# B&R Automation Studio project 8238 (part 7)

#### zz_KanlinkConfig.ab - Implementation code
```automation-basic
(********************************************************************
 * COPYRIGHT -- HP
 ********************************************************************
 * Program: zz_KanlinkConfig
 * File: zz_KanlinkConfig.ab
 * Author: treamsbottom
 * Created: September 07, 2012
 ********************************************************************
 * Implementation of program zz_KanlinkConfig
 ********************************************************************)
;Requirements
;From KGFramework
;	Libaries:
;		KgStdLib
;		KanLinkLib
;		mnParamLib
;	10ms Tasks:
;		hlKanLink
;	100ms Tasks:
;		svCPCache
;		mnEth
; When setting max connections for anything greater than 10
;the array decs will need changing. these are set by the constants HLKANLINK_MAX_CLIENTCONNS and HLKANLINK_MAX_SERVERCONNS in the frameworkshare
;Pkg_hlKanLink, KL_UserLib.Var
;----------------------------------------------------------------------------------------------------------------;
;-----21-1-2013..TR..Version A6 - First TestedVersion - Note Specials to run with Shuttle
;-----28-1-2013..TR..Version A7 - Remove Specials..Add option to send program and category number & Batch number.#
;-----03-03-2017..TR.Version A18 - Add "Advanced Connection Mode"
;-----07-06-2017 ..TR..Version A19 - Fix issues with sending empty bag date-- Remove reference to CAN[].Category -- Read all information from bag for consistency.
;-----------------------------------------------------------------------------------------------------------------
PROGRAM _INIT
	init := 0;
END_PROGRAM
PROGRAM _CYCLIC
;HLKANLINK_MAX_SERVERCONNS	;Declaration of max Server conns for KG Framework
;HLKANLINK_MAX_CLIENTCONNS	;Declaration of max Client conns for KG Framework
IF NOT init THEN
;Parameter Setup
;Global setting - Apply to all Kanlink Comms(Server,Client,OverView)
	Kanlink.GlobalSettings.TransferProgramCode 	= FALSE ; This transfers/Read the cat code to/from the bCustom area. Prg to/from sCategory
	Kanlink.GlobalSettings.TransferProgin_bCustom = FALSE ;This transfers/Read the Program code to/from the bCustom area. Category to/from sCategory
	Kanlink.GlobalSettings.UseBatchCode 		= TRUE	; Pass batch/SQL id
	Kanlink.GlobalSettings.BatchCodeTyp			= BatchTyp_UDINT  ;0 = UDINT, 1 = 16 byte unique (UDINT By default, extra code required for 16 byte )

;---------------------------------------------------------Batch Transfer Server---------------------------------------------------------------
;Server (Used to send data)		--------------------------- Variable = PT100
	Kanlink.Server.Enable = TRUE ; used to enable Server Comms
	Kanlink.Server.MaxConns	= 1 ; Number of Server connections
	 ; Start address of CAN variable
	;Address
	Kanlink.Server.IP[1].CommID = 1; //SDC1 R43
	Kanlink.Server.IP[1].Area 	= 3
	Kanlink.Server.IP[1].Adr 	= 11
;	Kanlink.Server.IP[1].AdvMode = FALSE // Use Advance mode- Pass in whole IP address as a string.
;	strcpy(ADR(Kanlink.Server.IP[1].AdrAdvMode),ADR("10.8.3.13"));
	Kanlink.Server.IP[1].CmdOpt = 0;

;	Kanlink.Server.IP[2].CommID = 2; //SDC2 R45
;	Kanlink.Server.IP[2].Area 	= 3
;	Kanlink.Server.IP[2].Adr 	= 12
;	Kanlink.Server.IP[2].CmdOpt = 0;
;
;	Kanlink.Server.IP[3].CommID = 3; //SDC3 R47
;	Kanlink.Server.IP[3].Area 	= 3
;	Kanlink.Server.IP[3].Adr 	= 13
;	Kanlink.Server.IP[3].CmdOpt = 0;
;
;	Kanlink.Server.IP[4].CommID = 4; //CDC8 R110
;	Kanlink.Server.IP[4].Area 	= 1
;	Kanlink.Server.IP[4].Adr 	= 12
;	Kanlink.Server.IP[4].CmdOpt = 0;
;
;	Kanlink.Server.IP[5].CommID = 5; //CDC9 R113
;	Kanlink.Server.IP[5].Area 	= 1
;	Kanlink.Server.IP[5].Adr 	= 2
;	Kanlink.Server.IP[5].CmdOpt = 0;
;
;	Kanlink.Server.IP[6].CommID = 6; //CDC6 R68
;	Kanlink.Server.IP[6].Area 	= 5
;	Kanlink.Server.IP[6].Adr 	= 15
;	Kanlink.Server.IP[6].CmdOpt = 0;
;
;	Kanlink.Server.IP[7].CommID = 7; //CDC7 R70
;	Kanlink.Server.IP[7].Area 	= 5
;	Kanlink.Server.IP[7].Adr 	= 16
;	Kanlink.Server.IP[7].CmdOpt = 0;
	;---------------------------------------------------------Batch transfer Client---------------------------------------------------------------
	;Client used to recieve data --------------------------- Variable = PTResp
	Kanlink.Client.Enable = TRUE ; used to enable Client Comms
	Kanlink.Client.MaxConns	= 2 ; Number of Client connections
	;Address

	//CSL1 r41
	Kanlink.Client.IP[1].CommID = 14	;//CSL1
	Kanlink.Client.IP[1].Area 	= 3
	Kanlink.Client.IP[1].Adr 	= 64
;	Kanlink.Client.IP[1].AdvMode = FALSE // Use Advance mode- Pass in whole IP address as a string.
;	strcpy(ADR(Kanlink.Client.IP[1].AdrAdvMode),ADR("10.8.4.20"));
	Kanlink.Client.IP[1].CmdOpt = 0

	//CSL2 r43
	Kanlink.Client.IP[2].CommID = 15	;//CSL2
	Kanlink.Client.IP[2].Area 	= 3
	Kanlink.Client.IP[2].Adr 	= 64
	Kanlink.Client.IP[2].CmdOpt = 1
;
;	//CSL1 r49
;	Kanlink.Client.IP[3].CommID = 11	;//CSL3
;	Kanlink.Client.IP[3].Area 	= 3
;	Kanlink.Client.IP[3].Adr 	= 62
;	Kanlink.Client.IP[3].CmdOpt = 0

;	//Sorting Rail
;	Kanlink.Client.IP[2].CommID = 4
;	Kanlink.Client.IP[2].Area 	= 3 ;Aero at sorting
;	Kanlink.Client.IP[2].Adr 	= 64
	;	Kanlink.Client.IP[1].AdvMode = FALSE // Use Advance mode- Pass in whole IP address as a string.
	;	strcpy(ADR(Kanlink.Client.IP[1].AdrAdvMode),ADR("10.8.4.20"));
;	Kanlink.Client.IP[2].CmdOpt = 1
;

;;---------------------------------------------------------Overview Server---------------------------------------------------------------
;	;------------------------------------------------Variable = STOverResp
;	;Use Overview Server.. SendData Data to Overview PLC - Only IP necessary - Client will request bag numbers.
	Kanlink.OverviewServer.Enable = FALSE
;	Kanlink.OverviewServer.MaxConns = 1
;
;	Kanlink.OverviewServer.IP[1].Area = 4
;	Kanlink.OverviewServer.IP[1].Adr = 21
;	Kanlink.OverviewServer.IP[1].AdvMode = FALSE
;	strcpy(ADR(Kanlink.OverviewServer.IP[1].AdrAdvMode),ADR("10.8.2.21"));
;
;	Kanlink.OverviewServer.IP[1].CmdOpt = 0
;;---------------------------------------------------------Overview Client---------------------------------------------------------------
;;------------------------------------------------Variable = STOverReq
;;Use Overview Client.. Recieve Data
	Kanlink.OverviewClient.Enable = FALSE
;	Kanlink.OverviewClient.MaxConns = 5
;	Kanlink.OverviewClient.CANOffset = 21
;;-----------PLC 1 - AERO SYSTEM
;	Kanlink.OverviewClient.StatusReg[1] = 951 ; D reg to map machine status for Tview.
;
;
;	Kanlink.OverviewClient.IP[1].Area = 3
;	Kanlink.OverviewClient.IP[1].Adr = 1	; To multiplex Edit KL_Overview
;	Kanlink.OverviewClient.IP[1].AdvMode = FALSE
;	strcpy(ADR(Kanlink.OverviewClient.IP[1].AdrAdvMode),ADR("10.8.3.1"));
;
;	Kanlink.OverviewClient.IP[1].CmdOpt = 0
;	//Batch data requested from Server
;	Kanlink.OverviewClient.InfoReq[1].wCntPositions = 6  ;Number of positions requested max 6 per request. If more than 6 set to 0 to multiplex...
;	Kanlink.OverviewClient.InfoReq[1].wNoOfPosition[0] = 1  ; Unqiue ID of data requested put all requests here if more than 6 the driver will multiplex the signals.
;	Kanlink.OverviewClient.InfoReq[1].wNoOfPosition[1] = 2	; There must be no gaps in the request numbers.	If not multiplexing, ensure index[6] = 0
;	Kanlink.OverviewClient.InfoReq[1].wNoOfPosition[2] = 3
;	Kanlink.OverviewClient.InfoReq[1].wNoOfPosition[3] = 4
;	Kanlink.OverviewClient.InfoReq[1].wNoOfPosition[4] = 5
;	Kanlink.OverviewClient.InfoReq[1].wNoOfPosition[5] = 6
;
;	//Bag number to map recieved data to.
;	Kanlink.OverviewClient.InfoResp[1].BagNum[0] = 501
;	Kanlink.OverviewClient.InfoResp[1].BagNum[1] = 502
;	Kanlink.OverviewClient.InfoResp[1].BagNum[2] = 503
;	Kanlink.OverviewClient.InfoResp[1].BagNum[3] = 504
;	Kanlink.OverviewClient.InfoResp[1].BagNum[4] = 505
;	Kanlink.OverviewClient.InfoResp[1].BagNum[5] = 506

;--------------------------------------------------------------END OF Configuration Code--------------------------------------------

;Check size of server and Client
	IF NOT Kanlink.Server.Enable THEN
		Kanlink.Server.MaxConns = 0
	ENDIF
	IF NOT Kanlink.Client.Enable THEN
		Kanlink.Client.MaxConns = 0
	ENDIF
	IF NOT Kanlink.OverviewServer.Enable THEN
		Kanlink.OverviewServer.MaxConns = 0
	ENDIF
	IF NOT Kanlink.OverviewClient.Enable THEN
		Kanlink.OverviewClient.MaxConns = 0
	ENDIF
	IF ((Kanlink.Server.MaxConns + Kanlink.OverviewServer.MaxConns) <= HLKANLINK_MAX_SERVERCONNS) THEN
		ServerDecOK = TRUE
	ELSE
		strcpy(ADR(Kanlink.ErrorString),"Declaration of HLKANLINK_MAX_SERVERCONNS not large enough")
		ServerDecOK = FALSE
	ENDIF
	IF ((Kanlink.Client.MaxConns + Kanlink.OverviewClient.MaxConns) <= HLKANLINK_MAX_CLIENTCONNS) THEN
		ClientDecOK = TRUE
	ELSE
		ClientDecOK = FALSE
		strcpy(ADR(Kanlink.ErrorString),"Declaration of HLKANLINK_MAX_CLIENTCONNS not large enough")
	ENDIF

	IF 	ServerDecOK AND ClientDecOK THEN

		;Server init
		IF Kanlink.Server.Enable THEN
			LOOP n = 1 TO Kanlink.Server.MaxConns DO
				;Build strings to pass to variable names, only required in a loop as index number changes.
				itoa(n,ADR(sn))	; put n into string
				strcpy(ADR(sReq),"PT100[");build string for variable name (request)
				strcat(ADR(sReq),ADR(sn))
				strcat(ADR(sReq),"].Req")
				strcpy(ADR(sResp),"PT100[");;build string for variable name (response)
				strcat(ADR(sResp),ADR(sn))
				strcat(ADR(sResp),"].Resp")
				IF Kanlink.Server.IP[n].AdvMode THEN
					IFhlKanLink.Parameter.Server[n].Adr = 0;
					IFhlKanLink.Parameter.Server[n].Area = 0
					IFhlKanLink.Parameter.Server[n].AdvMode := TRUE;
					strcpy(ADR(IFhlKanLink.Parameter.Server[n].AdrAdvMode),ADR(Kanlink.Server.IP[n].AdrAdvMode));
				ELSE
					IFhlKanLink.Parameter.Server[n].Adr = Kanlink.Server.IP[n].Adr ; Populate these arrays .
					IFhlKanLink.Parameter.Server[n].Area = Kanlink.Server.IP[n].Area
				ENDIF
				IFhlKanLink.Parameter.Server[n].Cmd = 1000 ; cmd from the server are always even
				IFhlKanLink.Parameter.Server[n].CmdOpt = Kanlink.Server.IP[n].CmdOpt
				IFhlKanLink.Parameter.Server[n].TimeOut = 1000 ;ms
				strcpy(ADR(IFhlKanLink.Parameter.Server[n].Name),"PT100") ; Diags Only
				strcpy(ADR(IFhlKanLink.Parameter.Server[n].sReq),ADR(sReq));"zzKanLink:PT100[0].Req")
				strcpy(ADR(IFhlKanLink.Parameter.Server[n].sResp),ADR(sResp));"zzKanLink:PT100[0].Resp")
			ENDLOOP
		ENDIF
		;Client Init
		IF Kanlink.Client.Enable THEN
			LOOP n = 1 TO Kanlink.Client.MaxConns DO
				itoa(n,ADR(sn))	; put n into string
				strcpy(ADR(sReq),"PTResp[");build string for variable name (request)
				strcat(ADR(sReq),ADR(sn))
				strcat(ADR(sReq),"].Req")
				strcpy(ADR(sResp),"PTResp[");;build string for variable name (response)
				strcat(ADR(sResp),ADR(sn))
				strcat(ADR(sResp),"].Resp")

				IF Kanlink.Client.IP[n].AdvMode THEN
					IFhlKanLink.Parameter.Client[n].Adr = 0;
					IFhlKanLink.Parameter.Client[n].Area = 0
					IFhlKanLink.Parameter.Client[n].AdvMode := TRUE;
					strcpy(ADR(IFhlKanLink.Parameter.Client[n].AdrAdvMode),ADR(Kanlink.Client.IP[n].AdrAdvMode));
				ELSE
					IFhlKanLink.Parameter.Client[n].Adr = Kanlink.Client.IP[n].Adr ; Populate these arrays .
					IFhlKanLink.Parameter.Client[n].Area = Kanlink.Client.IP[n].Area
				ENDIF
				IFhlKanLink.Parameter.Client[n].Cmd = 1000
				IFhlKanLink.Parameter.Client[n].CmdOpt = Kanlink.Client.IP[n].CmdOpt
				IFhlKanLink.Parameter.Client[n].CycleTime = 1000;ms
				strcpy(ADR(IFhlKanLink.Parameter.Client[n].Name),"PTResp")
				strcpy(ADR(IFhlKanLink.Parameter.Client[n].sReq),ADR(sReq))
				strcpy(ADR(IFhlKanLink.Parameter.Client[n].sResp),ADR(sResp))
			ENDLOOP
		ENDIF
		;Overview Server init
		;STOverResp[0] //Server sends batch data...
		IF Kanlink.OverviewServer.Enable THEN
			LOOP n = 1 TO Kanlink.OverviewServer.MaxConns DO
				;Build strings to pass to variable names, only required in a loop as index number changes.
				itoa(n,ADR(sn))	; put n into string
				strcpy(ADR(sReq),"STOverResp[");build string for variable name (request)
				strcat(ADR(sReq),ADR(sn))
				strcat(ADR(sReq),"].Req")
				strcpy(ADR(sResp),"STOverResp[");;build string for variable name (response)
				strcat(ADR(sResp),ADR(sn))
				strcat(ADR(sResp),"].Resp")

				Index = n + Kanlink.Server.MaxConns
				Kanlink.OverviewServer.IndexOffset = Kanlink.Server.MaxConns
				IF Kanlink.OverviewServer.IP[n].AdvMode THEN
					IFhlKanLink.Parameter.Server[Index].Adr = 0;
					IFhlKanLink.Parameter.Server[Index].Area = 0
					IFhlKanLink.Parameter.Server[Index].AdvMode := TRUE;
					strcpy(ADR(IFhlKanLink.Parameter.Server[Index].AdrAdvMode),ADR(Kanlink.OverviewServer.IP[n].AdrAdvMode));
				ELSE
					IFhlKanLink.Parameter.Server[Index].Adr = Kanlink.OverviewServer.IP[n].Adr ; Populate these arrays .
					IFhlKanLink.Parameter.Server[Index].Area = Kanlink.OverviewServer.IP[n].Area
				ENDIF

				IFhlKanLink.Parameter.Server[Index].Cmd = 1002 ;Batch Info Command
				IFhlKanLink.Parameter.Server[Index].CmdOpt = Kanlink.OverviewServer.IP[n].CmdOpt
				IFhlKanLink.Parameter.Server[Index].TimeOut = 1000 ;ms
				strcpy(ADR(IFhlKanLink.Parameter.Server[Index].Name),"STOverResp") ; Diags Only
				strcpy(ADR(IFhlKanLink.Parameter.Server[Index].sReq),ADR(sReq));"zzKanLink:STOverReq[0].Req")
				strcpy(ADR(IFhlKanLink.Parameter.Server[Index].sResp),ADR(sResp));"zzKanLink:STOverReq[0].Resp")

			ENDLOOP
		ENDIF

		;Kanlink OverView Client
		;STOverReq[0]// Client recieves batch data
		IF Kanlink.OverviewClient.Enable THEN
			LOOP n = 1 TO Kanlink.OverviewClient.MaxConns DO
				;Build strings to pass to variable names, only required in a loop as index number changes.
				itoa(n,ADR(sn))	; put n into string
				strcpy(ADR(sReq),"STOverReq[");build string for variable name (request)
				strcat(ADR(sReq),ADR(sn))
				strcat(ADR(sReq),"].Req")
				strcpy(ADR(sResp),"STOverReq[");;build string for variable name (response)
				strcat(ADR(sResp),ADR(sn))
				strcat(ADR(sResp),"].Resp")
				Index = n + Kanlink.Client.MaxConns
				Kanlink.OverviewClient.IndexOffset = Kanlink.Client.MaxConns

				IF Kanlink.OverviewClient.IP[n].AdvMode THEN
					IFhlKanLink.Parameter.Client[Index].Adr = 0;
					IFhlKanLink.Parameter.Client[Index].Area = 0
					IFhlKanLink.Parameter.Client[Index].AdvMode := TRUE;
					strcpy(ADR(IFhlKanLink.Parameter.Server[Index].AdrAdvMode),ADR(Kanlink.OverviewClient.IP[n].AdrAdvMode));
				ELSE
					IFhlKanLink.Parameter.Client[Index].Adr = Kanlink.OverviewClient.IP[n].Adr ; Populate these arrays .
					IFhlKanLink.Parameter.Client[Index].Area = Kanlink.OverviewClient.IP[n].Area
				ENDIF

				IFhlKanLink.Parameter.Client[Index].Cmd = 1002 ;Batch Info Command
				IFhlKanLink.Parameter.Client[Index].CmdOpt = Kanlink.OverviewClient.IP[n].CmdOpt
				IFhlKanLink.Parameter.Client[Index].CycleTime = 1000 ;ms
				strcpy(ADR(IFhlKanLink.Parameter.Client[Index].Name),"STOverReq") ; Diags Only
				strcpy(ADR(IFhlKanLink.Parameter.Client[Index].sReq),ADR(sReq));"zzKanLink:STOverResp[0].Req")
				strcpy(ADR(IFhlKanLink.Parameter.Client[Index].sResp),ADR(sResp));"zzKanLink:STOverResp[0].Resp")
			ENDLOOP
		ENDIF

		IFhlKanLink.in.xRestart = TRUE
		IFmnParam.Out.xParamOK = TRUE
		init = TRUE
		PT100 ; Variable that writes to the PT+ (Server)
		PTResp ; Variable that reads from PT+ (Client)
		STOverReq ;Variable used for the overview client
		STOverResp;Variable used for the overview server
	ENDIF//Server,client size OK
ENDIF//INIT

END_PROGRAM
```

#### zz_KanlinkConfig.var - Local variables
```iecst
(********************************************************************
 * COPYRIGHT -- HP
 ********************************************************************
 * Program: zz_KanlinkConfig
 * File: zz_KanlinkConfig.var
 * Author: treamsbottom
 * Created: September 07, 2012
 ********************************************************************
 * Local variables of program zz_KanlinkConfig
 ********************************************************************)
VAR
	UseServer : BOOL;
	UseClient : BOOL;
	init : BOOL;
	n : UINT;
	sn : STRING[5];
	sReq : STRING[20];
	sResp : STRING[20];
	ServerDecOK : BOOL;
	ClientDecOK : BOOL;
	Index : UINT;
END_VAR
```

### Program Logical/Standard/Kanlink/Kan_Driver (IEC, version 1.20.0) - *Kanlink Driver Server and Client

#### Kan_Driver.ab - Implementation code
```automation-basic
(********************************************************************
 * COPYRIGHT -- HP
 ********************************************************************
 * Program: Kan_Driver
 * File: Kan_Driver.ab
 * Author: treamsbottom
 * Created: September 07, 2012
 ********************************************************************
 * Implementation of program Kan_Driver
 ********************************************************************)
;----------------------------------------------------------------------------------------------------------------;
;-----21-1-2013..TR..Version A6 - First TestedVersion - Note 2 Specials in overview clien to run with Shuttle
;-----28-1-2013..TR..Version A7 - Remove Specials..Add option to send program and category number & Batch number.
;-----20-5-2014..TR..Version A12 - Fix ValidCat on DataValid
;-----09-01-2015..TR..Version A14 - Add Batching control
;-----02-08-2016 ..TR..Version A17 - Add Syncronous loading to Server Cmd 1000.. Use Comm[x].Transfer to watch for permission to unload.
;-----03-03-2017..TR.Version A18 - Add "Advanced Connection Mode"
;-----07-06-2017 ..TR..Version A19 - Fix issues with sending empty bag date-- Remove reference to Comm[].Category -- Read all information from bag for consistency.
;-----24-07-2018 ..TR -- Versioning Stopped Issues now tracked in GIT.
;-----27-10-2022 ..MS -- Added back Kanlink.OverviewServer and tested for BIT interface for Santorini Laundry.
;-----28-10-2022 ..MS -- Commented out comm.Program is no longer part of comm_type
;-----04-10-2023 ..MS -- Added CustomerStr and CategoryStr to comm_type to pass the string data read from kannlink

;-----------------------------------------------------------------------------------------------------------------
PROGRAM _INIT
	comm ACCESS ADR(Comm[0]);
END_PROGRAM
PROGRAM _CYCLIC
;Monitor State of supertrack (only send basic states now).
;IF (Kanlink.Server.Enable OR Kanlink.Client.Enable OR Kanlink.OverviewClient.Enable OR Kanlink.OverviewServer.Enable) THEN
;	IF SafetyZone[1].HaltSys THEN
;		SuperTrackState = KG_MACHINESTATE_EMERGENCYSTOP
;	ELSE
;		SuperTrackState = KG_MACHINESTATE_AUTOMATIC_RUN
;	ENDIF
;ENDIF
;--------------------------------------------------Kanlink Server Communication-----------------------------------------------------------------
IF Kanlink.Server.Enable THEN
	;Populate Batch Data
	LOOP n = 1 TO Kanlink.Server.MaxConns  DO
		IF (Kanlink.Server.IP[n].Adr > 0) THEN
			LOOP Index = 1 TO 1 DO ; Loop through each bag buffer
				comm ACCESS ADR(Comm[Kanlink.Server.IP[n].CommID]);
				IF (comm.Category > 0) THEN
					GetTimeStamp.enable = 1
					GetTimeStamp FUB DTGetTime()
					Batch[n].BatchData[Index].dtTimeStamp = GetTimeStamp.DT1
					;Make a string out OF CAT AND CUS
					length = itoa(comm.Category,ADR(myCategoryString));
					length = itoa(comm.Customer,ADR(myCustomerString));
					;copy Bag Data to KanLink Bag data type
;					IF Kanlink.GlobalSettings.TransferProgramCode THEN
;						Batch[n].BatchData[Index].sCategory = myProgramString
;						length = memcpy(ADR(Batch[n].BatchData[Index].bCustom),ADR(myCategoryString),12)
;					ELSE IF Kanlink.GlobalSettings.TransferProgin_bCustom THEN
;						Batch[n].BatchData[Index].sCategory = myCategoryString
;						length = memcpy(ADR(Batch[n].BatchData[Index].bCustom),ADR(myProgramString),12)
;					ELSE
						Batch[n].BatchData[Index].sCategory = myCategoryString
;					ENDIF
					IF Kanlink.GlobalSettings.UseBatchCode THEN
						IF Kanlink.GlobalSettings.BatchCodeTyp = BatchTyp_UDINT THEN
							;length = itoa(Bag[BagNumber].Mis,ADR(Batch[n].BatchData[Index].bBatchNo)) ; Convert to string
							length = memcpy(ADR(Batch[n].BatchData[Index].bBatchNo),ADR(comm.BatchID),4) ; Direct UDINT copy unreadble in KANLINK data.
						ELSE IF Kanlink.GlobalSettings.BatchCodeTyp = BatchTyp_16Byte THEN
							;Bag typ does not support this yet..
						ENDIF
					ELSE
						length = strcpy(ADR(Batch[n].BatchData[Index].bBatchNo),"")
					ENDIF
					Batch[n].BatchData[Index].bCntCustomers = 1
					Batch[n].BatchData[Index].wTotalWeight = comm.Weight;Summary weight of all Part Customers in the Bag, normally 1
					;First Customer in the Bag

					IF (comm.Batch_QtyRemaining <= 1) THEN
						Batch[n].BatchData[Index].PartBatch[0].sCustomNo = myCustomerString
						Batch[n].BatchData[Index].PartBatch[0].wCustomWeight =  comm.Batchpart[0].Wgt
					ELSE
						Batch[n].BatchData[Index].bCntCustomers = USINT(comm.Batch_QtyRemaining)
						LOOP t = 0 TO 7 DO
							length = itoa(comm.Batchpart[t].Customer,ADR(myCustomerString));
							Batch[n].BatchData[Index].PartBatch[t].sCustomNo = myCustomerString
							Batch[n].BatchData[Index].PartBatch[t].wCustomWeight = comm.Batchpart[t].Wgt
						ENDLOOP
					ENDIF
				ELSE
					strcpy(ADR(myCategoryString),ADR(""));
					strcpy(ADR(myCustomerString),ADR(""))
					strcpy(ADR(myProgramString),ADR(""));
					Batch[n].BatchData[Index].bCntCustomers = 0
					Batch[n].BatchData[Index].sCategory = myCategoryString
					length = strcpy(ADR(Batch[n].BatchData[Index].bCustom),"")
					length = strcpy(ADR(Batch[n].BatchData[Index].bBatchNo),"")
					Batch[n].BatchData[Index].wTotalWeight = 0 ;Summaray weight of all Part Customers in the Bag, normally 1
					LOOP t = 0 TO 7 DO
						Batch[n].BatchData[Index].PartBatch[t].sCustomNo = myCustomerString
						Batch[n].BatchData[Index].PartBatch[t].wCustomWeight = 0
					ENDLOOP
				ENDIF
				PT100[n].Resp.BatchData = Batch[n].BatchData[1] ; Only send first bag over KANLINK
			ENDLOOP

			; Handshake Signal Convert Comm into the KANLINK protocol
			;ValidCat = 	strcmp(ADR(comm.Category), "")
			//BagNumber = Kanlink.Server.BagNum[n].BagNums[1];
			IF (comm.Category > 0) THEN
				PT100[n].Resp.xHsDataValid = TRUE;
			ELSE
				PT100[n].Resp.xHsDataValid = FALSE
				PT100[n].Resp.xHsUnloading = FALSE
			ENDIF

			IF comm.BagReady THEN
				PT100[n].Resp.xHsReqForUnload = TRUE;
			ELSE
				PT100[n].Resp.xHsReqForUnload = FALSE;
			ENDIF

			comm.DropLoad 		= PT100[n].Req.xHreadyForLoad;
			comm.LoadDropped  	= PT100[n].Req.xHbatchReceived;
			PT100[n].Resp.wCntLoads = comm.Batch_QtyRemaining

			IF comm.DropLoad THEN
				PT100[n].Resp.xHsUnloading = TRUE
			ENDIF

			IF comm.HaltSys THEN
				PT100[n].Resp.wState = KG_MACHINESTATE_EMERGENCYSTOP
			ELSE
				PT100[n].Resp.wState = KG_MACHINESTATEX_AUTOMATIC_RUN
			ENDIF

			comm.Live = IFhlKanLink.Server[n].out.xConnected
			;Syncronous Loading.
			IF PT100[n].Req.xHreqCtrlTransfer THEN
				//Syncronous loading. Only allow unload when bit .x.x.x. is on
				PT100[n].Resp.xHsTransferRunning := PT100[n].Req.xHwaitingForTransfer;
			ELSE
				//Always give permission to unload..
				PT100[n].Resp.xHsTransferRunning := 1;
			ENDIF;
			comm.Transfer := PT100[n].Resp.xHsTransferRunning
		ENDIF
	ENDLOOP
ENDIF//ServerDriver
;--------------------------------------------------------Client Driver------------------------------------------------------------------
IF Kanlink.Client.Enable THEN
	LOOP n = 1 TO Kanlink.Client.MaxConns DO
		comm  ACCESS ADR(Comm[Kanlink.Client.IP[n].CommID])
		;Give Machine Ready
		PTResp[n].Req.xHready = TRUE
		PTResp[n].Req.bHcmdAutomatic = TRUE

		comm.BagReady = PTResp[n].Resp.xHsReqForUnload
		;Give ready to load when Ready
		PTResp[n].Req.xHreadyForLoad = comm.ReadyToLoad

		PTResp[n].Req.xHbatchReceived = comm.LoadRecieved
		;Send supertrack state
		IF comm.HaltSys THEN
			PTResp[n].Req.wHstate = KG_MACHINESTATE_EMERGENCYSTOP
		ELSE
			PTResp[n].Req.wHstate = KG_MACHINESTATEX_AUTOMATIC_RUN
		ENDIF
		;Check for Data Valid and unloading start.	then copy data to Comm Variable
		UnloadingPulse[n].CLK = (PTResp[n].Resp.xHsUnloading AND PTResp[n].Resp.xHsDataValid)
		UnloadingPulse[n] FUB R_TRIG()
		IF UnloadingPulse[n].Q THEN
;			IF Kanlink.GlobalSettings.TransferProgramCode THEN
;				comm.Program = USINT(atoi(ADR(PTResp[n].Resp.BatchData.sCategory)))
;				comm.Category = atoi(ADR(PTResp[n].Resp.BatchData.bCustom))
;			ELSE IF Kanlink.GlobalSettings.TransferProgin_bCustom THEN
;				comm.Program = USINT(atoi(ADR(PTResp[n].Resp.BatchData.bCustom)))
;				comm.Category = atoi(ADR(PTResp[n].Resp.BatchData.sCategory))
;			ELSE
				comm.Category = atoi(ADR(PTResp[n].Resp.BatchData.sCategory))
				comm.CategoryStr = PTResp[n].Resp.BatchData.sCategory
;			ENDIF
				comm.Customer = atoi(ADR(PTResp[n].Resp.BatchData.PartBatch[0].sCustomNo))
				comm.CustomerStr = PTResp[n].Resp.BatchData.PartBatch[0].sCustomNo
			comm.Weight = PTResp[n].Resp.BatchData.wTotalWeight
			IF Kanlink.GlobalSettings.UseBatchCode THEN
				IF Kanlink.GlobalSettings.BatchCodeTyp = BatchTyp_UDINT THEN
					length = memcpy(ADR(comm.BatchID),ADR(PTResp[n].Resp.BatchData.bBatchNo),4)
				ELSE IF Kanlink.GlobalSettings.BatchCodeTyp = BatchTyp_16Byte THEN
						;Bag typ does not support this yet..   KanLink_A19.var	Global variables	Directory="D:\Projects\Germany\SE8245_Wulf_Kiel\8245\bnr_plc\8245\Logical\Standard\Kanlink";Path="D:\Projects\Germany\SE8245_Wulf_Kiel\8245\bnr_plc\8245\Logical\Standard\Kanlink\KanLink_A19.var";Extension=".var";RefPath="";Reference="False"

				ENDIF
			ELSE
				comm.BatchID = 0
			ENDIF
		ENDIF

		comm.Unloading =  PTResp[n].Resp.xHsUnloading
		UnloadingFinishPLS[n].CLK = PTResp[n].Resp.xHsUnloading
		UnloadingFinishPLS[n] FUB F_TRIG()

		comm.UnloadFinished = UnloadingFinishPLS[n].Q
		;Comm Live
		comm.Live = IFhlKanLink.Client[n].out.xConnected
	ENDLOOP
ENDIF
;;---------------------------------------------------------------------------------------------Overview Client----------------------------------------
;IF Kanlink.OverviewClient.Enable THEN ; Collect data
;;------------------------------------------Build Request---------------------------------------------------
;
;	LOOP n = 1 TO Kanlink.OverviewClient.MaxConns DO
;
;
;		IF (CANOffset > 0) THEN
;			CANOffset = (Kanlink.OverviewClient.CANOffset - 1)
;			Comm[n+CANOffset].Live = IFhlKanLink.Client[n+Kanlink.OverviewClient.IndexOffset].out.xConnected
;			IF NOT Comm[n+CANOffset].Live THEN
;				D[Kanlink.OverviewClient.StatusReg[n]] = 0
;			ENDIF
;		ELSE
;			CANOffset = 0
;		ENDIF;
;
;		IF Kanlink.OverviewClient.InfoReq[n].wNoOfPosition[6] = 0 THEN ; do not multiplex data.
;			STOverReq[n].Req.wCntPositions = Kanlink.OverviewClient.InfoReq[n].wCntPositions;Number of Bags requested
;			DataOffset[n] = 0
;		ELSE
;
;			DataCount = 0
;			LOOP x = 0 TO 5 DO
;				IF (STOverReq[n].Req.wNoOfPosition[x] > 0) THEN
;					DataCount = DataCount + 1
;				ENDIF
;				IF DataCount > 5 THEN
;					DataCount = 6
;				ENDIF
;			ENDLOOP
;			STOverReq[n].Req.wCntPositions = DataCount;Number of Bags requested
;		ENDIF
;
;
;		LOOP x = 0 TO 5 DO
;			;datapositions requested
;			EXITIF ((DataOffset[n] + x) > HLKANLINK_MAX_OVERVIEW_DATA)
;
;			STOverReq[n].Req.wNoOfPosition[x] = Kanlink.OverviewClient.InfoReq[n].wNoOfPosition[x + DataOffset[n]]
;				;-----------------------------------------------Read Data----------------------------------
;			IF (STOverReq[n].Resp.wNoOfPositions[x] > 0) AND ((x <= STOverReq[n].Resp.wCntPositions) OR (STOverReq[n].Resp.wCntPositions = 0 )) THEN
;				IF (Kanlink.OverviewClient.InfoResp[n].BagNum[x + DataOffset[n]] > 0) THEN
;					IF Kanlink.OverviewClient.InfoReq[n].wNoOfPosition[x+DataOffset[n]] = STOverReq[n].Resp.wNoOfPositions[x] THEN
;					//	D[Kanlink.OverviewClient.StatusReg[n]] = STOverReq[n].Resp.wMachineState
;						BagIndex = Kanlink.OverviewClient.InfoResp[n].BagNum[x + DataOffset[n]]
;						IF Kanlink.GlobalSettings.TransferProgramCode THEN
;							Bag[BagIndex].Prg = USINT(atoi(ADR(STOverReq[n].Resp.BatchData[x].sCategory)))
;							Bag[BagIndex].Cat = atoi(ADR(STOverReq[n].Resp.BatchData[x].bCustom))
;						ELSE IF Kanlink.GlobalSettings.TransferProgin_bCustom THEN
;							Bag[BagIndex].Prg = USINT(atoi(ADR(STOverReq[n].Resp.BatchData[x].bCustom)))
;							Bag[BagIndex].Cat = atoi(ADR(STOverReq[n].Resp.BatchData[x].sCategory))
;						ELSE
;							Bag[BagIndex].Cat = atoi(ADR(STOverReq[n].Resp.BatchData[x].sCategory))
;						ENDIF
;						Bag[BagIndex].Cus = atoi(ADR(STOverReq[n].Resp.BatchData[x].PartBatch[0].sCustomNo)) ; Standard line of code..
;						Bag[BagIndex].Wgt = STOverReq[n].Resp.BatchData[x].PartBatch[0].wCustomWeight
;						IF Kanlink.GlobalSettings.UseBatchCode THEN
;							IF Kanlink.GlobalSettings.BatchCodeTyp = BatchTyp_UDINT THEN
;									length = memcpy(ADR(Bag[BagIndex].Mis),ADR(STOverReq[n].Resp.BatchData[x].bBatchNo),4)
;								ELSE IF	Kanlink.GlobalSettings.BatchCodeTyp = BatchTyp_16Byte THEN
;								;Not supported yet....
;							ENDIF
;						ELSE
;							Bag[BagIndex].Mis = 0
;						ENDIF
;					ENDIF
;				ENDIF
;			ENDIF
;		ENDLOOP
;		IF STOverReq[n].Resp.wNoOfPositions[0] = Kanlink.OverviewClient.InfoReq[n].wNoOfPosition[DataOffset[n]] THEN
;			DataOffset[n] = DataOffset[n] + 6
;		ELSE IF Kanlink.OverviewClient.InfoReq[n].wNoOfPosition[DataOffset[n]] = 0 THEN
;			DataOffset[n] = 0
;		ENDIF
;	ENDLOOP
;ENDIF
;
;---------------------------------------------------------------------------------------------Overview Server----------------------------------------
IF Kanlink.OverviewServer.Enable THEN
	LOOP n = 1 TO Kanlink.OverviewServer.MaxConns DO
		comm ACCESS ADR(Comm[Kanlink.OverviewServer.IP[n].CommID]);
		IF (STOverResp[n].Req.wCntPositions <= 6) THEN
			IF (STOverResp[n].Req.wCntPositions = 0) OR (STOverResp[n].Req.wCntPositions = 6) THEN
				NoOfDataRequested = 5
			ELSE
				NoOfDataRequested = STOverResp[n].Req.wCntPositions
			ENDIF
			LOOP x = 0 TO 0 DO
				IF x <= NoOfDataRequested THEN
					BagIndex = STOverResp[n].Req.wNoOfPosition[x]

					//STOverResp[n].Resp.wMachineState = SuperTrackState
					STOverResp[n].Resp.wNoOfPositions[x] = BagIndex
					STOverResp[n].Resp.wCntPositions = 	STOverResp[n].Req.wCntPositions
					//itoa(comm.Program,ADR(sProgram)) //Commented out as comm.Program is no longer part of comm_type
					itoa(comm.Category,ADR(sCategory))
					itoa(comm.Customer,ADR(sCustomer))
					itoa(comm.BatchID,ADR(sBatchID))
					STOverResp[n].Resp.BatchData[x].dtTimeStamp = GetTimeStamp.DT1
					IF Kanlink.GlobalSettings.TransferProgramCode THEN
						strcpy(ADR(STOverResp[n].Resp.BatchData[x].sCategory),ADR(sProgram))
						strcpy(ADR(STOverResp[n].Resp.BatchData[x].bCustom),ADR(sCategory))
					ELSE IF Kanlink.GlobalSettings.TransferProgin_bCustom THEN
						strcpy(ADR(STOverResp[n].Resp.BatchData[x].sCategory),ADR(sCategory))
						strcpy(ADR(STOverResp[n].Resp.BatchData[x].bCustom),ADR(sProgram))
					ELSE
						strcpy(ADR(STOverResp[n].Resp.BatchData[x].sCategory),ADR(sCategory))
					ENDIF
					IF Kanlink.GlobalSettings.UseBatchCode THEN
						IF Kanlink.GlobalSettings.BatchCodeTyp = BatchTyp_UDINT THEN
							length = memcpy(ADR(STOverResp[n].Resp.BatchData[x].bBatchNo),ADR(comm.BatchID),4)
						ELSE IF Kanlink.GlobalSettings.BatchCodeTyp = BatchTyp_UDINT THEN
							strcpy(ADR(STOverResp[n].Resp.BatchData[x].bBatchNo),ADR(sBatchID))
						ENDIF
					ELSE
						strcpy(ADR(STOverResp[n].Resp.BatchData[x].bBatchNo),"")
					ENDIF
					strcpy(ADR(STOverResp[n].Resp.BatchData[x].PartBatch[0].sCustomNo),ADR(sCustomer))
					STOverResp[n].Resp.BatchData[x].wTotalWeight = comm.Weight			//11.11.2019 BIT to show weight
					STOverResp[n].Resp.BatchData[x].PartBatch[0].wCustomWeight = comm.Weight
				ELSE
					STOverResp[n].Resp.wNoOfPositions[x] = 0
					STOverResp[n].Resp.BatchData[x].dtTimeStamp = 0
					strcpy(ADR(STOverResp[n].Resp.BatchData[x].sCategory),"")
					strcpy(ADR(STOverResp[n].Resp.BatchData[x].bCustom),"")
					strcpy(ADR(STOverResp[n].Resp.BatchData[x].bBatchNo),"")
					strcpy(ADR(STOverResp[n].Resp.BatchData[x].PartBatch[0].sCustomNo),"")
					STOverResp[n].Resp.BatchData[x].wTotalWeight = 0 //11.11.2019 BIT to show weight
					STOverResp[n].Resp.BatchData[x].PartBatch[0].wCustomWeight = 0
				ENDIF
			ENDLOOP
		ENDIF
	ENDLOOP
ENDIF

END_PROGRAM
```

#### Kan_Driver.var - Local variables
```iecst
(********************************************************************
 * COPYRIGHT -- HP
 ********************************************************************
 * Program: Kan_Driver
 * File: Kan_Driver.var
 * Author: treamsbottom
 * Created: September 07, 2012
 ********************************************************************
 * Local variables of program Kan_Driver
 ********************************************************************)
VAR
	n : UINT;
	Index : UINT;
	BagNumber : UINT;
	GetTimeStamp : DTGetTime;
	length : UDINT;
	myCategoryString : STRING[11];
	myCustomerString : STRING[11];
	UnloadingPulse : ARRAY[0..HLKANLINK_MAX_CLIENTCONNS] OF R_TRIG;
	UnloadingFinishPLS : ARRAY[0..HLKANLINK_MAX_CLIENTCONNS] OF F_TRIG;
	SuperTrackState : USINT;
	x : UINT;
	BagIndex : UINT;
	sCustomer : STRING[11];
	sCategory : STRING[11];
	sBatchID : STRING[16];
	NoOfDataRequested : UINT;
	DataOffset : ARRAY[0..HLKANLINK_MAX_CLIENTCONNS] OF UINT;
	DataCount : UINT;
	myProgramString : STRING[11];
	sProgram : STRING[11];
	t : UINT;
	comm : REFERENCE TO Comm_typ;
END_VAR
```

### Package Logical/Standard/Kanlink/KGFramework - Standard-Packages

### Package Logical/Standard/Kanlink/KGFramework/Pkg_KGStandard - Kannegiesser Standards

### Stat.var - Package variables
```iecst
(********************************************************************
 * COPYRIGHT -- Herbert Kannegiesser GmbH
 ********************************************************************
 * Package: Pkg_KGStandard
 * File: Stat.var
 * Author: hunholz
 * Created: March 07, 2012
 ********************************************************************
 * Variables of package Pkg_KGStandard
 ********************************************************************)
VAR CONSTANT
	KG_STAT_OK : UINT := 0;
	KG_STAT_BUSY : UINT := 65535;
END_VAR
```

### utfNames.typ - Package data types
```iecst
(********************************************************************
 * COPYRIGHT -- Microsoft
 ********************************************************************
 * Package: Pkg_KGStandard
 * File: utfNames.typ
 * Author: hunholz
 * Created: June 29, 2011
 ********************************************************************
 * Data types of package Pkg_KGStandard
 ********************************************************************)
(*Abgeleitete Datentypen dürfen nicht als Parameter verwendet
werden, da der Parameter-Manager bzw. die B&R-System-Funktion
dann den Datentypen nicht ermitteln kann!!!*)

TYPE
	utfName31_typ :WSTRING[31];
	utfName15_typ :WSTRING[15];
END_TYPE
```

### kgbom.var - Package variables
```iecst
(********************************************************************
 * COPYRIGHT -- Herbert Kannegiesser GmbH
 ********************************************************************
 * Package: Pkg_KGStandard
 * File: kgbom.var
 * Author: hunholz
 * Created: December 20, 2011
 ********************************************************************
 * Variables of package Pkg_KGStandard
 ********************************************************************)
VAR
	KGBOM : ARRAY[0..1] OF USINT := [16#FF,16#FE];
END_VAR
```

### Library Logical/Standard/Kanlink/KGFramework/Pkg_KGStandard/KGstdLib (IEC) - Kannegiesser Hilfsfunktionen
Depends on: astime, AsIODiag, Ethernet, AsBrStr, DataObj, AsArLog

#### KGstdLib_History.txt
```
1.02.0	NEU: kgGetMacAdress, kgGetBatchNoLong, kgGetBatchNoUnique
	    Library umbenannt in KGstdLib
		Umgestellt auf AS 3.0.90
1.16.2  Bugfix kgCheckDo
		Abhängigkeiten ergänzt
1.17.0	kgUnitconfREALtoDisplay erweitert um Einheitenstring
```

#### KGstdLib_Doc.txt
```
KGstdLib-Dokumentation
======================

----------------------
Abgeleitete Datentypen
----------------------

	MAC_type	USINT[0..5]
	GUID_type	USINT[0..15]

---------------
Konvertierungen
---------------

kgitoa_udint
------------

	Beschreibung:
	------------
	Wandelt eine UDINT-Variable in einen String

	Rückgabewert
	------------

				UDINT		0	-	OK

	VAR_INPUT
	---------

		num		UDINT		Zu wandelnder Zahlenwert

	VAR_IN_OUT
	----------

		str		STRING[11]	Ergebnis

kgatoi_udint
------------

	Beschreibung:
	------------
	Wandelt einen STRING in einen UDINT-Wert

	Rückgabewert
	------------

				UDINT		0	-	OK
							1	-	zu viele Ziffern
							2	-	ungültiges Zeichen
							3	-	Außerhalb des Wertebereichs

	VAR_INPUT
	---------

		str		STRING[11]	Zu wandelnder String

	VAR_IN_OUT
	----------

		num		UDINT		Ergebnis

kgatoi_uint
------------

	Beschreibung:
	------------
	Wandelt einen STRING in einen UINT-Wert

	Rückgabewert
	------------

				UINT		0	-	OK
							1	-	zu viele Ziffern
							2	-	ungültiges Zeichen
							3	-	Außerhalb des Wertebereichs

	VAR_INPUT
	---------

		str		STRING[5	Zu wandelnder String

	VAR_IN_OUT
	----------

		num		UINT		Ergebnis

---------------
Postennummern
---------------

kgNextBatchNoLong
-----------------

	Beschreibung:
	-------------
	Erzeugt eine eindeutige Postennummer im Format UDINT
	Es sollte immer sichergestellt sein, dass die Uhr der SPS gestellt ist.

	Verwendete Libraries:
	---------------------

		astime

	VAR_INPUT
	---------

		Enable	BOOL	Eine neue Postennummer wird immer mit der positiven Flanke von Enable erzeugt.
						D.h. der FB muss zwischenzeitlich mit Enable := FALSE aufgerufen werden.

		Group	USINT	Bis zu 8 Maschinen in einem Systemverbund können Postennummern erzeugen. Dazu
						benötigt die Maschine eine eindeutige Gruppennummer von 0 .. 7.

	VAR_IN_OUT
	----------

		BatchNo	UDINT	Die Postennummer baut immer auf die vorhergehende Nummer auf. Darum wird dem
						FB die alte Nummer übergeben und die neue Nummer zurückgeliefert.

	VAR_OUTPUT
	----------

		Status	UINT	0 		- OK
						1		- Am Tag sind nur 4096 Postennummern je Gruppe möglich. Diese Maximalgrenze wurde überschritten.
						65534	- Enable = FALSE

kgGetBatchNoUnique
------------------

	Beschreibung:
	-------------
	Erzeugt eine eindeutige, 16 Byte lange Postennummer im Format GUID
	Es sollte immer sichergestellt sein, dass die Uhr der SPS gestellt ist.

	Verwendete Libraries:
	---------------------

		astime

	VAR_INPUT
	---------

		Enable	BOOL		Eine neue Postennummer wird immer mit der positiven Flanke von Enable erzeugt.
							D.h. der FB muss zwischenzeitlich mit Enable := FALSE aufgerufen werden.

		Mac		MAC_type	In eine GUID wird immer die MAC-Adresse der Steuerung kodiert. Die MAC-Adresse
							muss im Init_Up mit kgGetMacAdress ausgelesen werden.

	VAR_OUTPUT
	----------

		BatchNo	GUID_type	GUID

		Status	UINT		0 		- OK
							65534 	- Enable = FALSE

---------------
Sonstiges
---------------

kgGetMacAdress
--------------

	Beschreibung:
	------------
	Ermittelt die MAC-Adresse der onboard Ethernetschnittstelle

	Verwendete Libraries:
	---------------------

		AsBrStr, Netlink, Ethernet

	VAR_INPUT
	---------

		Enable	BOOL	keine Funktion

	VAR_OUTPUT
	----------

		Mac		MAC_type	MAC-Adresse

		Status	UINT		0 - OK
							Stati von ETHxinfo und GetEthPort
```

#### KG_Cmd.typ - Package data types
```iecst
(********************************************************************
 * COPYRIGHT -- Herbert Kannegiesser GmbH
 ********************************************************************
 * File: KG_Cmd.typ
 * Author: hunholz
 * Created: Feb 29, 2012
 ********************************************************************
 * Global data types of KGFramework
 ********************************************************************)

TYPE
	KG_Cmd_typ : 	STRUCT
		Response : KG_CmdResponse_typ; (*Wird vom verantwortlichen SPS-Package beschrieben*)
		Request : KG_CmdRequest_typ; (*Wird nur von "außerhalb" beschrieben*)
	END_STRUCT;
	KG_CmdRequest_typ : 	STRUCT
		Command : KG_Command_typ; (*Kommando mit Attributen. Zusätzliche Attribute werden über eine zusätzliche Struktur übergeben.*)
	END_STRUCT;
	KG_CmdResponse_typ : 	STRUCT
		wCmdStatus : UINT; (*Rückgabewert. 0 - NoCommand, 1..59999 - Rückgabe des Kommandowertes bei erfolgreichem Abschluss, 60000..65534 - Fehler, 65535 - Busy*)
		wLockStatus : UINT; (*0 - Kommandokanal ist frei, Clientnummer des Clients, der den Kommandokanal blockiert hat*)
	END_STRUCT;
	KG_Command_typ : 	STRUCT
		wCommand : UINT; (*0 - kein Kommando, 1..59999 - Gültige Kommandonummer*)
		lData0 : UDINT; (*beliebig, entsprechend des Kommandos*)
		lData1 : UDINT; (*beliebig, entsprechend des Kommandos*)
	END_STRUCT;
END_TYPE
```

#### Stat.typ - Package data types
```iecst
(********************************************************************
 * COPYRIGHT -- Microsoft
 ********************************************************************
 * Package: Pkg_KGStandard
 * File: State.typ
 * Author: hunholz
 * Created: September 20, 2011
 ********************************************************************
 * Data types of package Pkg_KGStandard
 ********************************************************************)

TYPE
	Stat_typ : 	STRUCT
		wStatus : UINT;
		sStatus : STRING[127];
	END_STRUCT;
END_TYPE
```

#### KGstdLib.typ - Exported data types
```iecst
(********************************************************************
 * COPYRIGHT -- Microsoft
 ********************************************************************
 * Library: KGstd
 * File: KGstd.typ
 * Author: hunholz
 * Created: June 23, 2011
 ********************************************************************
 * Data types of library KGstd
 ********************************************************************)

TYPE
	MAC_type :ARRAY[0..5]OF USINT;
	GUID_type :ARRAY[0..15]OF USINT;
	KG_ErrLog_typ : 	STRUCT
		wErrorNo : UINT;
		lAttr1 : UDINT;
		lAttr2 : UDINT;
	END_STRUCT;
END_TYPE
```

#### kgMachineState.typ - Package data types
```iecst
(********************************************************************
 * COPYRIGHT -- Herbert Kannegiesser GmbH
 ********************************************************************
 * Package: Pkg_KGStandard
 * File: kgMachineState.typ
 * Author: hunholz
 * Created: April 11, 2012
 ********************************************************************
 * Data types of package Pkg_KGStandard
 ********************************************************************)

TYPE
	kgMachineState_enum :
		(
		msOFF := 0, (*Machine turned off*)
		msEmergency_Stop := 1, (*Emergency stop*)
		msSafe := 2, (*Safety stop*)
		msFault := 3, (*Fault*)
		msFaultWaitQuit := 4, (*Fault, waiting for acknowledge*)
		msService := 5, (*Service*)
		msAutomatic := 6, (*Automatic run*)
		msStop := 7, (*Stop*)
		msStandby := 8, (*Automatic wait (Standby)*)
		msStandbyWaitQuit := 9, (*Automatic wait for manuel action*)
		msWarning := 10, (*Automatic warning*)
		msAuto_Dryer_Heating := 30,
		msAuto_Dryer_Cooldown := 31,
		msAuto_Dryer_Clean_Filter := 32,
		msAuto_Dryer_Afterrung := 33,
		msAuto_Dryer_Cleaningfan_Running := 34,
		msAuto_Conv_Fwd := 40,
		msAuto_Conv_Fwd2nd := 41,
		msAuto_Conv_Rev := 42,
		msAuto_Conv_Rev2nd := 43
		);
END_TYPE
```

#### kgMachinetyp.typ - Package data types
```iecst
(********************************************************************
 * COPYRIGHT -- Herbert Kannegiesser GmbH
 ********************************************************************
 * Package: Pkg_KGStandard
 * File: kgMachinetyp.typ
 * Author: hunholz
 * Created: January 27, 2012
 ********************************************************************
 * Data types of package Pkg_KGStandard
 ********************************************************************)
(**********************************)
(*Maschinentypen, -gruppen*)
(***********************************)

TYPE
	kgMachinetypeW3_typ :
		(
		kgW3LOADSYSTEM := 0,
		kgW3WASHER := 10,
		kgW3WETSHUTTLE := 30,
		kgW3EXTRACTOR := 40,
		kgW3EXTRACTOR2 := 50, (*behind a WETSHUTTLE*)
		kgW3CONVEYOR := 60,
		kgW3DRYER := 70,
		kgW3SHAKER := 110, (*"Entsander"*)
		kgW3SINGLEWASHER := 120, (*FA+*)
		kgW3PROCESS := 150, (*EMS, Silo-Tank*)
		kgW3IFBOX := 160,
		kgW3DEVICE := 180, (*Camera, Printer*)
		kgW3SERVER := 202,
		kgW3PCSTATION := 210,
		kgW3BIT := 230,
		kgW3NOTDEFINED := 255
		);
END_TYPE
```

#### KG_Cmd.var - Package variables
```iecst
(********************************************************************
 * COPYRIGHT -- Herbert Kannegiesser GmbH
 ********************************************************************
 * Package: Pkg_KGStandard
 * File: KG_Cmd.var
 * Author: hunholz
 * Created: March 05, 2012
 ********************************************************************
 * Variables of package Pkg_KGStandard
 ********************************************************************)
VAR CONSTANT
	KG_CMD_NOCOMMAND : UINT := 0; (*Kein Kommando*)
	KG_CMD_GETLOCK : UINT := 59998; (*Lock für xxxCmdAd Struktur anfordern*)
	KG_CMD_RELEASELOCK : UINT := 59999; (*Lock für xxxCmdAd Struktur freigeben*)
	KG_CMDSTAT_NOTREADY : UINT := 65529; (*Nicht bereit*)
	KG_CMDSTAT_INVALID_PARAMETER : UINT := 65530; (*Mindestens ein Parameter ist nicht zulässig*)
	KG_CMDSTAT_GETLOCKFAILED : UINT := 65531; (*Lock konnte nicht gesetzt werden*)
	KG_CMDSTAT_RELEASELOCKFAILED : UINT := 65532; (*Lock darf nicht freigegeben werden.*)
	KG_CMDSTAT_NOTVALID : UINT := 65533; (*Kommando ungültig*)
	KG_CMDSTAT_BUSY : UINT := 65535; (*Kommando wird bearbeitet*)
END_VAR
```

#### KGstdLib.var - Exported constants
```iecst
(********************************************************************
 * COPYRIGHT -- Microsoft
 ********************************************************************
 * Library: KGstd
 * File: KGstd.var
 * Author: hunholz
 * Created: June 23, 2011
 ********************************************************************
 * Constants of library KGstd
 ********************************************************************)
VAR CONSTANT
	KG_AUTH_LOCKED : USINT := 0;
	KG_AUTH_OPERATOR : USINT := 1;
	KG_AUTH_TECHNICIAN : USINT := 2;
	KG_AUTH_KGTECHNICIAN : USINT := 3;
	KG_AUTH_ADMIN : USINT := 4;
	KG_AUTH_NOACK : USINT := 255;
END_VAR
(*Errors*)
VAR CONSTANT
	KG_ERR_RB_NOREAD : UINT := 1;
	KG_ERR_RB_POINTER : UINT := 2;
	KG_ERR_RB_WRITEPOINTER : UINT := 3;
	KG_ERR_RB_READPOINTER : UINT := 4;
	KG_ERR_RB_STARTPOINTER : UINT := 5;
	KG_ERR_RB_LOCPOINTER : UINT := 6;
	KG_ERR_RB_SIZE : UINT := 7;
	KG_ERR_GETETHPORT_IFSTRING : UINT := 21;
	KG_ERR_GETETHPORT_ADRIF : UINT := 22;
	KG_ERR_WRONGSIZES : UINT := 30;
	KG_INFO_DO_NEW : UINT := 31;
	KG_ERR_NULPOINTER : UINT := 40;
	KG_ERR_NULLSTRING : UINT := 41;
END_VAR
(*RB Modus für kgRBloc*)
VAR CONSTANT
	KG_RB_LOC_MODE_ABSOLUTE : USINT := 0;
	KG_RB_LOC_MODE_FROMSTART : USINT := 1;
	KG_RB_LOC_MODE_FROMEND : USINT := 2;
END_VAR
(*CPU Identifier*)
VAR CONSTANT
	KG_CPU_X20CP1484 : UDINT := 16#23A5;
	KG_CPU_X20CP1484_1 : UDINT := 16#AABE;
	KG_CPU_X20CP3484 : UDINT := 16#23A6;
	KG_CPU_X20CP3484_1 : UDINT := 16#AABF;
	KG_CPU_X20CP1486 : UDINT := 16#2164;
	KG_CPU_X20CP3486 : UDINT := 16#1F19;
	KG_CPU_X20CP3585 : UDINT := 16#C3AF;
	KG_CPU_X20CP1584 : UDINT := 16#C370;
	KG_CPU_X20CP1586 : UDINT := 16#C3B0;
	KG_CPU_PP420_1043_75 : UDINT := 16#23BD;
	KG_CPU_PP65_0571_P74 : UDINT := 16#A964;
	KG_CPU_CTT_11 : UDINT := 16#A2BC;
	KG_CPU_PCT_03 : UDINT := 16#A7DD;
	KG_CPU_PCT_04 : UDINT := 16#B399;
END_VAR
(*Module Identifier*)
VAR CONSTANT
	KG_MODULE_NO : UDINT := 16#0000;
	KG_MODULE_X20DI9371 : UDINT := 16#1B95;
	KG_MODULE_X20DO9322 : UDINT := 16#1B9A;
	KG_MODULE_X20BR9300 : UDINT := 16#1BC1;
	KG_MODULE_X20PS2100 : UDINT := 16#1BBF;
	KG_MODULE_4PP065IF231 : UDINT := 16#B0BB;
	KG_MODULE_X20IF1072 : UDINT := 16#1F20;
	KG_MODULE_X20IF2772 : UDINT := 16#1F25;
	KG_MODULE_X20BT9400 : UDINT := 16#A238;
	KG_MODULE_X67DM1321 : UDINT := 16#1311;
END_VAR
(*Units*)
VAR CONSTANT
	KG_UNIT_METRIC : USINT := 0;
	KG_UNIT_US : USINT := 1;
END_VAR
```

#### kgMachineState.var - Package variables
```iecst
(********************************************************************
 * COPYRIGHT -- Herbert Kannegiesser GmbH
 ********************************************************************
 * Package: Pkg_KGStandard
 * File: kgMachineState.var
 * Author: hunholz
 * Created: January 27, 2012
 ********************************************************************
 * Variables of package Pkg_KGStandard
 ********************************************************************)
VAR CONSTANT
	KG_MACHINESTATE_OFF : USINT := 16#0; (*Machine is turned off*)
	KG_MACHINESTATE_EMERGENCYSTOP : USINT := 16#1; (*Emergency stop*)
	KG_MACHINESTATE_SAFESTOP : USINT := 16#2; (*Safe stop*)
	KG_MACHINESTATE_FAULT : USINT := 16#3; (*Fault*)
	KG_MACHINESTATE_FAULT_GONE : USINT := 16#4; (*Fault, wait for acknowledge*)
	KG_MACHINESTATE_SERVICE : USINT := 16#5; (*Service*)
	KG_MACHINESTATE_AUTOMATIC_RUN : USINT := 16#6; (*Automatic Run*)
	KG_MACHINESTATE_STOP : USINT := 16#7; (*Stop*)
	KG_MACHINESTATE_WAIT_AUTOMATIC : USINT := 16#8; (*Automatic Wait (Standby)*)
	KG_MACHINESTATE_WAIT_MAN : USINT := 16#9; (*Automatic Wait for manual action*)
	KG_MACHINESTATE_WARNING : USINT := 16#A; (*Automatic Warning*)
END_VAR
(*Special states for dryer*)
VAR CONSTANT
	KG_MACHINESTATE_DRY_HEATING : USINT := 16#1E; (*Automatic heating*)
	KG_MACHINESTATE_DRY_COOLDOWN : USINT := 16#1F; (*Automatic cooldown*)
	KG_MACHINESTATE_DRY_CLEAN_FILTER : USINT := 16#20; (*Automatic clean filter*)
	KG_MACHINESTATE_DRY_AFTERRUN : USINT := 16#21; (*Automatic afterrun*)
	KG_MACHINESTATE_DRY_FAN_CLEAN : USINT := 16#22; (*Automatic running cleaning fan*)
END_VAR
(*Special states for conveyor*)
VAR CONSTANT
	KG_MACHINESTATE_CONV_FWD : USINT := 16#28; (*Automatic running forward*)
	KG_MACHINESTATE_CONV_FWD2 : USINT := 16#29; (*Automatic running forward 2nd speed*)
	KG_MACHINESTATE_CONV_REV : USINT := 16#2A; (*Automatic running reverse*)
	KG_MACHINESTATE_CONV_REV2 : USINT := 16#2B; (*Automatic running reverse 2nd speed*)
END_VAR
(*ENHANCED STATES*)
VAR CONSTANT
	KG_MACHINESTATEX_OFF : UINT := 16#100; (*Machine is turned off*)
	KG_MACHINESTATEX_EMERGENCYSTOP : UINT := 16#101; (*Emergency stop*)
	KG_MACHINESTATEX_SAFESTOP : UINT := 16#102; (*Safe stop*)
	KG_MACHINESTATEX_FAULT : UINT := 16#103; (*Fault*)
	KG_MACHINESTATEX_FAULT_GONE : UINT := 16#104; (*Fault, wait for acknowledge*)
	KG_MACHINESTATEX_SERVICE : UINT := 16#105; (*Service*)
	KG_MACHINESTATEX_AUTOMATIC_RUN : UINT := 16#6; (*Automatic Run*)
	KG_MACHINESTATEX_STOP : UINT := 16#107; (*Stop*)
	KG_MACHINESTATEX_WAIT_AUTOMATIC : UINT := 16#208; (*Automatic Wait (Standby)*)
	KG_MACHINESTATEX_WAIT_MAN : UINT := 16#209; (*Automatic Wait for manual action*)
	KG_MACHINESTATEX_WARNING : UINT := 16#A; (*Automatic Warning*)
END_VAR
(*Special states for dryer*)
VAR CONSTANT
	KG_MACHINESTATEX_DRY_HEATING : UINT := 16#1E; (*Automatic heating*)
	KG_MACHINESTATEX_DRY_COOLDOWN : UINT := 16#1F; (*Automatic cooldown*)
	KG_MACHINESTATEX_DRY_CLEAN_FILTE : UINT := 16#20; (*Automatic clean filter*)
	KG_MACHINESTATEX_DRY_AFTERRUN : UINT := 16#21; (*Automatic afterrun*)
	KG_MACHINESTATEX_DRY_FAN_CLEAN : UINT := 16#22; (*Automatic running cleaning fan*)
END_VAR
(*Special states for conveyor*)
VAR CONSTANT
	KG_MACHINESTATEX_CONV_FWD : UINT := 16#28; (*Automatic running forward*)
	KG_MACHINESTATEX_CONV_FWD2 : UINT := 16#29; (*Automatic running forward 2nd speed*)
	KG_MACHINESTATEX_CONV_REV : UINT := 16#2A; (*Automatic running reverse*)
	KG_MACHINESTATEX_CONV_REV2 : UINT := 16#2B; (*Automatic running reverse 2nd speed*)
END_VAR
```

#### KGstdLib.fun - Exported functions and function blocks
```iecst
(********************************************************************
 * COPYRIGHT -- Microsoft
 ********************************************************************
 * Library: KGstd
 * File: KGstd.fun
 * Author: hunholz
 * Created: June 23, 2011
 ********************************************************************
 * Functions and function blocks of library KGstd
 ********************************************************************)

FUNCTION_BLOCK kgGetEthPort (*Returns the CPUs ethernet port as string*)
	VAR_INPUT
		enable : BOOL;
		adrIF : UDINT;
	END_VAR
	VAR_OUTPUT
		status : UINT;
	END_VAR
	VAR
		_bStep : USINT;
		DiagCreateInfo_CPU : DiagCreateInfo;
		DiagGetNumInfo_CPU : DiagGetNumInfo;
		DiagDisposeInfo_CPU : DiagDisposeInfo;
		_xReady : BOOL;
	END_VAR
END_FUNCTION_BLOCK

FUNCTION kgitoa_udint : UINT (*Wandelt UDINT Werte in einen String*)
	VAR_INPUT
		num : UDINT;
	END_VAR
	VAR_IN_OUT
		str : STRING[11];
	END_VAR
	VAR
		_num : UDINT;
		_digit : UDINT;
		_sdigit : STRING[1];
		_bdigit : REFERENCE TO USINT;
	END_VAR
END_FUNCTION

FUNCTION kgatoi_udint : UINT (*String in UDINT wandeln*)
	VAR_INPUT
		str : STRING[11];
	END_VAR
	VAR_IN_OUT
		num : UDINT;
	END_VAR
	VAR
		_len : UINT;
		_result : UINT;
		_sdigit : STRING[1];
		_bdigit : REFERENCE TO USINT;
		_mul : UDINT;
		_digit : UDINT;
		_i : INT;
	END_VAR
END_FUNCTION

FUNCTION kgatoi_uint : UINT (*atoi für UINT mit Fehlermeldung*)
	VAR_INPUT
		str : STRING[11];
	END_VAR
	VAR_IN_OUT
		num : UINT;
	END_VAR
	VAR
		_result : UINT;
		_len : INT;
		_sdigit : STRING[1];
		_bdigit : REFERENCE TO USINT;
		_mul : UINT;
		_i : INT;
		_digit : USINT;
	END_VAR
END_FUNCTION

FUNCTION_BLOCK kgNextBatchNoLong (*Generiert eine neue Postennummer*)
	VAR_INPUT
		Enable : BOOL; (*Positive Flanke erzeugt neue Nummer*)
		Group : USINT; (*0..7*)
	END_VAR
	VAR_OUTPUT
		Status : UINT; (*0 : OK, 1 : Maximale Anzahl möglicher Nummern pro Tag erreich, B&R Werte*)
		BatchNo : UDINT;
	END_VAR
	VAR
		_bOldYear : USINT;
		_bOldMonth : USINT;
		_bOldDay : USINT;
		DTStrucGetTime : DTStructureGetTime;
		_dtStruc : DTStructure;
		_bGroup : USINT;
		_wNo : UINT;
		_bStep : USINT;
		_diBatchNo : DatObjInfo;
		_pBatchNo : REFERENCE TO UDINT;
		_dwBatchNo : DatObjWrite;
		_dcBatchNo : DatObjCreate;
		zzEdge00000 : BOOL;
	END_VAR
END_FUNCTION_BLOCK

FUNCTION_BLOCK kgGetMacAdress (*Nur im Init-Up aufrufen*)
	VAR_INPUT
		Enable : BOOL;
	END_VAR
	VAR_OUTPUT
		Mac : MAC_type;
		Status : UINT;
	END_VAR
	VAR
		_gep : kgGetEthPort;
		_sIF : STRING[23];
		_exi : ETHxinfo;
		_bMAC : MAC_type;
	END_VAR
END_FUNCTION_BLOCK

FUNCTION_BLOCK kgGetBatchNoUnique (*Batchnummer als Unique Identifier 16 Byte*)
	VAR_INPUT
		Enable : BOOL;
		Mac : MAC_type;
	END_VAR
	VAR_OUTPUT
		BatchNo : GUID_type;
		Status : UINT;
	END_VAR
	VAR
		DTGetTime_0 : DTGetTime;
		_time : TIME;
	END_VAR
END_FUNCTION_BLOCK

FUNCTION kgBatchNoToUDINT : UDINT (*Extrahiere aus GUID ein UDINT*)
	VAR_INPUT
		GUID : GUID_type;
	END_VAR
	VAR
		_udint : REFERENCE TO UDINT;
	END_VAR
END_FUNCTION

FUNCTION_BLOCK kgUSINT16toGUID (*Konvertiere USINT-Array to GUID_typ*)
	VAR_INPUT
		usintarray : ARRAY[0..15] OF USINT;
	END_VAR
	VAR_OUTPUT
		GUID : GUID_type;
	END_VAR
END_FUNCTION_BLOCK

FUNCTION_BLOCK kgGUIDtoSTRING (*GUID-String erzeugen*)
	VAR_INPUT
		GUID : GUID_type;
	END_VAR
	VAR_OUTPUT
		sOut : STRING[36];
	END_VAR
	VAR
		usintarray : REFERENCE TO ARRAY[0..15] OF USINT;
		_StringArray : REFERENCE TO ARRAY[0..36] OF USINT;
		_Ptr : INT;
		_i : INT;
		_b : USINT;
	END_VAR
END_FUNCTION_BLOCK

FUNCTION_BLOCK kgLogLine (*Logzeile mit zwei numerischen Variablen erzeugen*)
	VAR_INPUT
		sLoglineTemplate : STRING[127];
		lAttr1 : UDINT;
		lAttr2 : UDINT;
	END_VAR
	VAR_OUTPUT
		sLogline : STRING[127];
		pLogline : UDINT;
	END_VAR
	VAR
		_iPos1 : INT;
		_iPos2 : INT;
		_iCrs : INT;
		sValue : STRING[11];
		_sTemp : STRING[127];
	END_VAR
END_FUNCTION_BLOCK

FUNCTION_BLOCK kgArLogWrite (*Checks ident on > 0 and formats string with two numbers*)
	VAR_INPUT
		enable : BOOL;
		ident : UDINT;
		logLevel : UDINT;
		errornr : UDINT;
		text : STRING[127];
		var1 : UDINT;
		var2 : UDINT;
	END_VAR
	VAR_OUTPUT
		status : UINT;
	END_VAR
	VAR
		_AsArLogWrite : AsArLogWrite;
		_kgLogLine : kgLogLine;
	END_VAR
END_FUNCTION_BLOCK

FUNCTION_BLOCK kgRBinsert (*Insert any entry into a ringbuffer*)
	VAR_INPUT
		pEntry : UDINT;
		lLenEntry : UDINT;
		doIdent : UDINT;
		doLen : UDINT;
	END_VAR
	VAR_OUTPUT
		wStatus : UINT;
	END_VAR
	VAR_IN_OUT
		wPtrStart : UINT;
		wPtrWrite : UINT;
		wPtrRead : UINT;
	END_VAR
	VAR
		doWrite : DatObjWrite;
		_lRBlen : UDINT;
		_wPtrMax : UINT;
	END_VAR
END_FUNCTION_BLOCK

FUNCTION_BLOCK kgRBread (*Reads one entry and moves the readpointer*)
	VAR_INPUT
		pEntry : UDINT;
		lLenEntry : UDINT;
		doIdent : UDINT;
		doLen : UDINT;
		wPtrStart : UINT;
		wPtrWrite : UINT;
	END_VAR
	VAR_OUTPUT
		wStatus : UINT;
	END_VAR
	VAR_IN_OUT
		wPtrRead : UINT;
	END_VAR
	VAR
		doRead : DatObjRead;
		_lRBlen : UDINT;
		_wPtrMax : UINT;
	END_VAR
END_FUNCTION_BLOCK

FUNCTION_BLOCK kgRBloc (*Free Readpointer access*)
	VAR_INPUT
		pEntry : UDINT;
		lLenEntry : UDINT;
		doIdent : UDINT;
		doLen : UDINT;
		wPtrStart : UINT;
		wPtrWrite : UINT;
		wPtrLoc : UINT;
		bMode : USINT; (*Lese relativ zum Start- oder Schreibzeiger*)
	END_VAR
	VAR_OUTPUT
		wStatus : UINT;
	END_VAR
	VAR
		doRead : DatObjRead;
		_lRBlen : UDINT;
		_wPtrMax : UINT;
		_wPtrLoc : UINT;
		_wActLen : UINT;
	END_VAR
END_FUNCTION_BLOCK

FUNCTION kgGUIDisZero : BOOL (*Prüfen, ob alle 16 Byte der GUID 0 sind.*)
	VAR_INPUT
		GUID : GUID_type;
	END_VAR
	VAR
		_bGUID : REFERENCE TO ARRAY[0..15] OF USINT;
		_i : USINT;
	END_VAR
END_FUNCTION

FUNCTION_BLOCK kgRBcreate (*Erzeuge Datenobjekt für Ringbuffer*)
	VAR_INPUT
		sName : STRING[10]; (*Name des Datenobjekts*)
		bMemType : USINT; (*Speichertyp*)
		wCntEntry : UINT; (*Mindestanzahl der RB_Einträge*)
		lLenEntry : UDINT; (*Länge des einzelnen Eintrags*)
	END_VAR
	VAR_OUTPUT
		doIdent : UDINT; (*Identifier des Datenobjekts*)
		doLen : UDINT; (*Länge des Datenobjekts*)
		wStatus : UINT; (*Status*)
		pDatObjMem : UDINT;
	END_VAR
	VAR_IN_OUT
		wPtrWrite : UINT; (*Schreibzeiger*)
		wPtrRead : UINT; (*Lesezeiger*)
		wPtrStart : UINT; (*Startzeiger*)
	END_VAR
	VAR
		_diRB : DatObjInfo;
		_dcRB : DatObjCreate;
		_ddRB : DatObjDelete;
	END_VAR
END_FUNCTION_BLOCK

FUNCTION_BLOCK kgRBbulkloc (*Lese mehrere Einträge gleichzeitig in ein Array*)
	VAR_INPUT
		pEntry : UDINT; (*Zeiger auf den Zielbereich*)
		lLenEntry : UDINT; (*Länge eines Eintrags*)
		wCntEntry : UINT; (*Anzahl Einträge*)
		doIdent : UDINT;
		doLen : UDINT;
		wPtrStart : UINT;
		wPtrWrite : UINT;
		wPtrLoc : UINT;
		bMode : USINT;
	END_VAR
	VAR_OUTPUT
		wStatus : UINT;
		wCntLoc : UINT;
	END_VAR
	VAR
		_lRBlen : UDINT;
		_wPtrMax : UINT;
		_wActLen : UINT;
		_wPtrLoc : UINT;
		_i : UINT;
		_doRead : DatObjRead;
	END_VAR
END_FUNCTION_BLOCK

FUNCTION kgGetLineNumberW3 : USINT (*Maschinennummer und -typ aus Stationsadresse berechnen*)
	VAR_INPUT
		Station : USINT;
		pMachineType : UDINT;
	END_VAR
	VAR
		_MachineType : REFERENCE TO kgMachinetypeW3_typ;
	END_VAR
END_FUNCTION

FUNCTION_BLOCK kgInitBatchNoLong (*Legt ggf. Datenobjekt zum Speichern der laufenden Postennummer an*)
	VAR_INPUT
		Enable : BOOL;
	END_VAR
	VAR_OUTPUT
		Status : UINT;
	END_VAR
	VAR
		_bStep : USINT;
		_diBatchNo : DatObjInfo;
		_dcBatchNo : DatObjCreate;
		_BatchNo : UDINT;
	END_VAR
END_FUNCTION_BLOCK

FUNCTION kgGetMachineAdressW3 : USINT (*Ermittelt die Maschinenadresse aus Liniennummer und Maschinentyp*)
	VAR_INPUT
		LineNumber : USINT;
		MachineType : kgMachinetypeW3_typ;
	END_VAR
	VAR
		_diMachineType : REFERENCE TO DINT;
	END_VAR
END_FUNCTION

FUNCTION_BLOCK kgCheckDo (*Prüfe auf Datenobjekt und erzeuge es ggf. neu*)
	VAR_INPUT
		Enable : BOOL;
		pName : UDINT;
		MinLen : UDINT;
		NomLen : UDINT;
		Create : BOOL;
		MemType : USINT;
	END_VAR
	VAR_OUTPUT
		doId : UDINT;
		doMem : UDINT;
		doLen : UDINT;
		Status : UINT;
	END_VAR
	VAR
		_wStep : UINT;
		_doInfo : DatObjInfo;
		_xReady : BOOL;
		_doDelete : DatObjDelete;
		_doCreate : DatObjCreate;
	END_VAR
END_FUNCTION_BLOCK

FUNCTION kgXOR : USINT (*XOR über Byte-Feld*)
	VAR_INPUT
		pMem : UDINT; (*Speicher*)
		wLen : UINT; (*Länge*)
		bInit : USINT; (*Startwert*)
		pStatus : UDINT; (*Status*)
		pWordResult : UDINT;
	END_VAR
	VAR
		_wDynStatus : REFERENCE TO UINT;
		_xStatusOk : BOOL;
		_bMem : REFERENCE TO ARRAY[1..65535] OF USINT;
		_xWordResultOk : BOOL;
		_bWordResult : REFERENCE TO ARRAY[0..1] OF USINT;
		_i : UINT;
	END_VAR
END_FUNCTION

FUNCTION kgUnitconfREALtoDisplay : REAL (*Wandelt Wert entsprechend der Unit*)
	VAR_INPUT
		Value : REAL;
		Unit : UINT;
		LocUnit : USINT;
		pDigits : UDINT;
		pUnit : UDINT;
	END_VAR
	VAR
		lDigits : UDINT;
		sUnit : STRING[11];
	END_VAR
END_FUNCTION

FUNCTION kgUnitconfDisplayToREAL : REAL (*Wandelt Wert entsprechend der Unit*)
	VAR_INPUT
		Display : REAL;
		Unit : UINT;
		LocUnit : USINT;
	END_VAR
END_FUNCTION

FUNCTION kgGetProgdata : UINT (*Read Programdata from a dataobject*)
	VAR_INPUT
		sBaseName : STRING[11];
		wProgNo : UINT;
		wProgMaxNo : UINT;
		pMem : UDINT;
		lSize : UDINT;
	END_VAR
	VAR
		_sIndex : STRING[5];
		_sIndex1 : STRING[5];
		_sName : STRING[16];
		_diProg : DatObjInfo;
	END_VAR
END_FUNCTION

FUNCTION kgSignalLight : BOOL
	VAR_INPUT
		xClock : BOOL;
		wStatus : UINT;
	END_VAR
	VAR_IN_OUT
		xGreen : BOOL;
		xYellow : BOOL;
		xRed : BOOL;
	END_VAR
END_FUNCTION
```

#### kgitoa_udint.st - Wandelt UDINT in String
```iecst
(********************************************************************
 * COPYRIGHT -- Microsoft
 ********************************************************************
 * Library: KGstd
 * File: kgitoa_udint.st
 * Author: hunholz
 * Created: June 23, 2011
 ********************************************************************
 * Implementation of library KGstd
 ********************************************************************)

(* Wandelt UDINT in String *)
FUNCTION kgitoa_udint

	_num := num;
	str := '';
	_sdigit := '0';
	_bdigit ACCESS ADR(_sdigit);

	REPEAT

		_digit := _num MOD 10;

		_bdigit := 48 + UDINT_TO_USINT(_digit);
		str := INSERT(str,_sdigit,0);

		_num := _num / 10;

	UNTIL
		_num = 0
	END_REPEAT;

	kgitoa_udint := 0;

END_FUNCTION
```

#### kgatoi_udint.st - String in UDINT wandeln
```iecst
(********************************************************************
 * COPYRIGHT -- Microsoft
 ********************************************************************
 * Library: KGstd
 * File: kgatoi_udint.st
 * Author: hunholz
 * Created: June 23, 2011
 ********************************************************************
 * Implementation of library KGstd
 ********************************************************************)

(* String in UDINT wandeln *)
FUNCTION kgatoi_udint

	num := 0;

	_result := 0;

	_len := LEN(str);

	_sdigit := '0';
	_bdigit ACCESS ADR(_sdigit);

	_mul := 1;

	// Ist String generell zu lang ?
	IF _len > 10 THEN

		_result := 1;

	ELSIF _len > 0 THEN

		FOR _i := _len TO 1 BY -1 DO

			_sdigit := MID(str,1, _i);

			// Auf ungültiges Zeiche prüfen
			IF (_bdigit < 48 OR _bdigit > 57) THEN
				_result := 2;
				num := 0;
				EXIT;
			ELSE
				_digit := _bdigit - 48;
			END_IF

			// Auf Wertüberlauf prüfen
			IF _len = 10 AND _i = 1 THEN

				IF _digit > 4 OR (_digit = 4 AND num > 294967295) THEN
					_result := 3;
					num := 0;
					EXIT;
				END_IF

			END_IF

			num := num + (_digit * _mul);

			IF (_i <> 1) THEN
				_mul := _mul * 10;
			END_IF

		END_FOR

	END_IF

	kgatoi_udint := _result;

END_FUNCTION
```

#### kgatoi_uint.st - atoi für UINT mit Fehlermeldung
```iecst
(********************************************************************
 * COPYRIGHT -- Microsoft
 ********************************************************************
 * Library: KGstd
 * File: kgatoi_uint.st
 * Author: hunholz
 * Created: June 28, 2011
 ********************************************************************
 * Implementation of library KGstd
 ********************************************************************)

(* atoi für UINT mit Fehlermeldung *)
FUNCTION kgatoi_uint

	num := 0;

	_result := 0;

	_len := LEN(str);

	_sdigit := '0';
	_bdigit ACCESS ADR(_sdigit);

	_mul := 1;

	// Ist String generell zu lang ?
	IF _len > 5 THEN

		_result := 1;

	ELSIF _len > 0 THEN

		FOR _i := _len TO 1 BY -1 DO

			_sdigit := MID(str,1, _i);

			// Auf ungültiges Zeiche prüfen
			IF (_bdigit < 48 OR _bdigit > 57) THEN
				_result := 2;
				num := 0;
				EXIT;
			ELSE
				_digit := _bdigit - 48;
			END_IF

			// Auf Wertüberlauf prüfen
			IF _len = 5 AND _i = 1 THEN

				IF _digit > 6 OR (_digit = 6 AND num > 5535) THEN
					_result := 3;
					num := 0;
					EXIT;
				END_IF

			END_IF

			num := num + (_digit * _mul);

			IF (_i <> 1) THEN
				_mul := _mul * 10;
			END_IF

		END_FOR

	END_IF

	kgatoi_uint := _result;

END_FUNCTION
```

#### kgInitBatchNoLong.st - Legt ggf. Datenobjekt zum Speichern der laufenden Postennummer an
```iecst
(********************************************************************
 * COPYRIGHT -- Herbert Kannegiesser GmbH
 ********************************************************************
 * Library: KGstdLib
 * File: kgInitBatchNoLong.st
 * Author: hunholz
 * Created: January 31, 2012
 ********************************************************************
 * Implementation of library KGstdLib
 ********************************************************************)

(* Legt ggf. Datenobjekt zum Speichern der laufenden Postennummer an *)
FUNCTION_BLOCK kgInitBatchNoLong

	IF Enable AND _bStep = 0 THEN
		_bStep := 1;
	END_IF

	IF _bStep = 1 AND NOT Enable THEN
		_bStep := 0;
	END_IF

	CASE _bStep OF

		0: // Enable ist FALSE

			Status := ERR_FUB_ENABLE_FALSE;

		1: // Enable ist TRUE

			_diBatchNo(enable := TRUE, pName := ADR('_BatchNo'));

			IF _diBatchNo.status = doERR_MODULNOTFOUND THEN

				Status := ERR_FUB_BUSY;

				_bStep := 2;

			ELSE

				Status := _diBatchNo.status;

			END_IF

		2: // Create DO

			_dcBatchNo.enable := TRUE;
			_dcBatchNo.len := SIZEOF(_BatchNo);
			_dcBatchNo.MemType := doUSRROM;
			_dcBatchNo.pName := ADR('_BatchNo');

			_dcBatchNo();

			Status := _dcBatchNo.status;

			IF _dcBatchNo.status <> ERR_FUB_BUSY THEN
				_bStep := 1;
			END_IF

	END_CASE

END_FUNCTION_BLOCK
```

#### kgNextBatchNoLong.st - Generiert eine neue Postennummer bei positiver Flanke von Enable
```iecst
(********************************************************************
 * COPYRIGHT -- Microsoft
 ********************************************************************
 * Library: KGstd
 * File: kgNextBatchNoLong.st
 * Author: hunholz
 * Created: July 19, 2011
 * Changed: Feb 15, 2012
 ********************************************************************
 * Implementation of library KGstd
 ********************************************************************)

(* Generiert eine neue Postennummer *)
FUNCTION_BLOCK kgNextBatchNoLong

	IF EDGEPOS(Enable) THEN
		IF _bStep = 0 THEN
			_bStep := 1;
		END_IF
	END_IF

	IF _bStep = 255 AND NOT Enable THEN
		_bStep := 0;
	END_IF

	CASE _bStep OF

		0: // Enable ist FALSE

			Status := ERR_FUB_ENABLE_FALSE;

		1: // Enable ist TRUE

			_diBatchNo(enable := TRUE, pName := ADR('_BatchNo'));

			IF _diBatchNo.status = ERR_OK THEN

				_pBatchNo ACCESS _diBatchNo.pDatObjMem;

				// Datum der aktuellen Postennummer extrahieren
				_bOldYear := UDINT_TO_USINT( SHR( (_pBatchNo AND 16#003F8000) ,15));
				_bOldMonth := UDINT_TO_USINT( SHR( (_pBatchNo AND 16#03C00000) , 22));
				_bOldDay := UDINT_TO_USINT( SHR( (_pBatchNo AND 16#7C000000) ,26));
				_bGroup := UDINT_TO_USINT( SHR( (_pBatchNo AND 16#00007000) ,12));
				_wNo := UDINT_TO_UINT( _pBatchNo AND 16#00000FFF );

				DTStrucGetTime.enable := TRUE;
				DTStrucGetTime.pDTStructure := ADR(_dtStruc);
				DTStrucGetTime();

				IF (_bGroup <> Group MOD 8 ) THEN
					_bGroup := Group MOD 8;
					_wNo := 0;
				END_IF

				IF (_bOldDay <> _dtStruc.day) OR (_bOldMonth <> _dtStruc.month) OR (_bOldYear <> UINT_TO_USINT(_dtStruc.year MOD 2000) ) THEN
					_bOldDay := _dtStruc.day;
					_bOldMonth := _dtStruc.month;
					_bOldYear := UINT_TO_USINT(_dtStruc.year MOD 2000);
					_wNo := 0;
				END_IF

				IF _wNo = 4095 THEN

					Status := 1;

				ELSE

					_wNo := _wNo + 1;

					BatchNo := 0;
					BatchNo := BatchNo OR SHL(USINT_TO_UDINT(_bOldDay),26);
					BatchNo := BatchNo OR SHL(USINT_TO_UDINT(_bOldMonth),22);
					BatchNo := BatchNo OR SHL(USINT_TO_UDINT(_bOldYear),15);
					BatchNo := BatchNo OR SHL(USINT_TO_UDINT(_bGroup),12);
					BatchNo := BatchNo OR UINT_TO_UDINT(_wNo);

					_dwBatchNo(enable := TRUE, ident := _diBatchNo.ident, len := SIZEOF(BatchNo), Offset := 0, pSource := ADR(BatchNo));

					Status := _dwBatchNo.status;

				END_IF

				_bStep := 255;	// Fertig

			ELSE

				_bStep := 2;	// Datenobjekt anlegen

				Status := ERR_FUB_BUSY;

			END_IF

		2:	// Datenobjekt anlegen

			_dcBatchNo.enable := TRUE;
			_dcBatchNo.len := SIZEOF(BatchNo);
			_dcBatchNo.MemType := doUSRROM;
			_dcBatchNo.pName := ADR('_BatchNo');

			_dcBatchNo();

			Status := _dcBatchNo.status;

			IF _dcBatchNo.status = ERR_OK THEN
				_bStep := 1;

				Status := ERR_FUB_BUSY;

			ELSIF _dcBatchNo.status <> ERR_FUB_BUSY THEN

				Status := _dcBatchNo.status;
				BatchNo := 0;
				_bStep := 255;

			END_IF

		255:	// Fertig

			_diBatchNo(enable := TRUE, pName := ADR('_BatchNo'));

			IF _diBatchNo.status = ERR_OK THEN

				_pBatchNo ACCESS _diBatchNo.pDatObjMem;
				BatchNo := _pBatchNo;

			ELSE

				_bStep := 2;	// Datenobjekt anlegen

				Status := ERR_FUB_BUSY;

				BatchNo := 0;

			END_IF

	END_CASE

END_FUNCTION_BLOCK
```

#### kgGetMacAdress.st
```iecst
(********************************************************************
 * COPYRIGHT -- Microsoft
 ********************************************************************
 * Library: KGstd
 * File: kgGetMacAdress.st
 * Author: hunholz
 * Created: July 19, 2011
 ********************************************************************
 * Implementation of library KGstd
 ********************************************************************)

(* TODO: Add your comment here *)
FUNCTION_BLOCK kgGetMacAdress

	IF Enable THEN

		// MAC-Adresse initialisieren
		brsmemset(ADR(Mac),0,SIZEOF(Mac));

		// Ermittle den Ethernet-Devicestring aus der CPU-ID
		// Siehe Library Netlink

		_gep.enable := TRUE;
		_gep.adrIF := ADR(_sIF);

		REPEAT

			_gep();

		UNTIL

			_gep.status <> ERR_FUB_BUSY

		END_REPEAT

		// Lese die MAC-Adresse aus

		IF _gep.status = 0 THEN

			_exi.enable := TRUE;
			_exi.pDevice := ADR(_sIF);

			_exi();

			_bMAC := _exi.mac;

			Status := _exi.status;

			IF Status = 0 THEN

				Mac := _bMAC;

			END_IF

		ELSE

			Status := _gep.status;

		END_IF

	ELSE

		Status := ERR_FUB_ENABLE_FALSE;

	END_IF

END_FUNCTION_BLOCK
```

#### kgGetBatchNoUnique.st - Batchnummer als Unique Identifier 16 Byte, wenn Enable = TRUE
```iecst
(********************************************************************
 * COPYRIGHT -- Microsoft
 ********************************************************************
 * Library: KGstd
 * File: kgGetBatchNoUnique.st
 * Author: hunholz
 * Created: July 19, 2011
 * Changed: February 15, 2012
 ********************************************************************
 * Implementation of library KGstd
 ********************************************************************)

(* Batchnummer als Unique Identifier 16 Byte *)
FUNCTION_BLOCK kgGetBatchNoUnique

	Status := ERR_OK;

	brsmemset(ADR(BatchNo),0,SIZEOF(BatchNo));

	IF Enable THEN

		DTGetTime_0(enable := TRUE);

		_time := clock_ms();

		brsmemcpy(ADR(BatchNo[0]),ADR(DTGetTime_0.DT1), 4);
		brsmemcpy(ADR(BatchNo[4]),ADR(_time), 2);
		BatchNo[6] := 16#10;
		brsmemcpy(ADR(BatchNo[7]),ADR(_time)+2, 1);
		BatchNo[8] := 16#50;
		brsmemcpy(ADR(BatchNo[9]),ADR(_time)+3, 1);
		brsmemcpy(ADR(BatchNo[10]), ADR(Mac[0]), 6);

	ELSE

		Status := ERR_FUB_ENABLE_FALSE;

	END_IF

END_FUNCTION_BLOCK
```

#### kgBatchNoToUDINT.st - Extrahiere aus GUID ein UDINT
```iecst
(********************************************************************
 * COPYRIGHT -- Herbert Kannegiesser GmbH
 ********************************************************************
 * Library: KGstdLib
 * File: kgBatchNoToUDINT.st
 * Author: hunholz
 * Created: November 17, 2011
 ********************************************************************
 * Implementation of library KGstdLib
 ********************************************************************)

(* Extrahiere aus GUID ein UDINT *)
FUNCTION kgBatchNoToUDINT

	_udint ACCESS ADR(GUID);

	kgBatchNoToUDINT := _udint;

END_FUNCTION
```

#### kgUSINT16toGUID.st - Konvertiere USINT-Array to GUID_typ
```iecst
(********************************************************************
 * COPYRIGHT -- Herbert Kannegiesser GmbH
 ********************************************************************
 * Library: KGstdLib
 * File: kgUSINT16toGUID.st
 * Author: hunholz
 * Created: November 17, 2011
 ********************************************************************
 * Implementation of library KGstdLib
 ********************************************************************)

(* Konvertiere USINT-Array to GUID_typ *)
FUNCTION_BLOCK kgUSINT16toGUID

	brsmemcpy(ADR(GUID), ADR(usintarray), SIZEOF(GUID));

END_FUNCTION_BLOCK
```

#### kgGUIDtoSTRING.st - GUID-String erzeugen
```iecst
(********************************************************************
 * COPYRIGHT -- Herbert Kannegiesser GmbH
 ********************************************************************
 * Library: KGstdLib
 * File: kgGUIDtoSTRING.st
 * Author: hunholz
 * Created: November 17, 2011
 ********************************************************************
 * Implementation of library KGstdLib
 ********************************************************************)

(* GUID-String erzeugen *)
FUNCTION_BLOCK kgGUIDtoSTRING

	usintarray ACCESS ADR(GUID);

	brsmemset(ADR(sOut), 0, SIZEOF(sOut));

	_StringArray ACCESS ADR(sOut);

	_Ptr := 0;

	FOR _i := 0 TO 15 DO

		_b := (usintarray[_i] / 16);

		IF _b < 10 THEN
			_StringArray[_Ptr] := _b + 48;
		ELSE
			_StringArray[_Ptr] := _b + 65;
		END_IF

		_Ptr := _Ptr + 1;

		_b := (usintarray[_i] MOD 16);

		IF _b < 10 THEN
			_StringArray[_Ptr] := _b + 48;
		ELSE
			_StringArray[_Ptr] := _b + 65;
		END_IF

		_Ptr := _Ptr + 1;

		IF _i = 3 OR _i = 5 OR _i = 7 OR _i = 9 THEN

			_StringArray[_Ptr] := 45; // '-'
			_Ptr := _Ptr + 1;

		END_IF

	END_FOR

END_FUNCTION_BLOCK
```

#### kgLogLine.st - Logzeile mit zwei numerischen Variablen erzeugen
```iecst
(********************************************************************
 * COPYRIGHT -- Herbert Kannegiesser GmbH
 ********************************************************************
 * Library: KGstdLib
 * File: kgLogLine.st
 * Author: hunholz
 * Created: December 19, 2011
 ********************************************************************
 * Implementation of library KGstdLib
 ********************************************************************)

(* Logzeile mit zwei numerischen Variablen erzeugen *)
FUNCTION_BLOCK kgLogLine

	sLogline := '';
	pLogline := ADR(sLogline);

	IF LEN(sLoglineTemplate) > 0 THEN

		_iPos1 := FIND(sLoglineTemplate,'{##AttrVar1}');
		_iPos2 := FIND(sLoglineTemplate,'{##AttrVar2}');
		_iCrs := 1;

		IF (_iPos1 > 0) AND (_iPos2 = 0 OR _iPos1 < _iPos2) THEN

			_sTemp := MID(sLoglineTemplate, _iPos1 - _iCrs, _iCrs);
			sLogline := CONCAT(sLogline, _sTemp);
			_iCrs := _iPos1 + 12;
			_iPos1 := 0;

			brsitoa(lAttr1, ADR(sValue));
			sLogline := CONCAT(sLogline, sValue);

		END_IF

		IF (_iPos2 > 0) AND (_iPos1 = 0 OR _iPos2 < _iPos1) THEN

			_sTemp := MID(sLoglineTemplate, _iPos2 - _iCrs, _iCrs);
			sLogline := CONCAT(sLogline, _sTemp);
			_iCrs := _iPos2 + 12;
			_iPos2 := 0;

			brsitoa(lAttr2, ADR(sValue));
			sLogline := CONCAT(sLogline, sValue);

		END_IF

		IF (_iPos1 > 0) THEN

			_sTemp := MID(sLoglineTemplate, _iPos1 - _iCrs, _iCrs);
			sLogline := CONCAT(sLogline, _sTemp);
			_iCrs := _iPos1 + 12;

			brsitoa(lAttr1, ADR(sValue));
			sLogline := CONCAT(sLogline, sValue);

		END_IF

		_sTemp := RIGHT(sLoglineTemplate, LEN(sLoglineTemplate)-_iCrs+1);
		sLogline := CONCAT(sLogline, _sTemp);

	END_IF

END_FUNCTION_BLOCK
```

#### kgArLogWrite.st - Checks ident on > 0 and formats string with two numbers
```iecst
(********************************************************************
 * COPYRIGHT -- Herbert Kannegiesser GmbH
 ********************************************************************
 * Library: KGstdLib
 * File: kgArLogWrite.st
 * Author: hunholz
 * Created: December 19, 2011
 ********************************************************************
 * Implementation of library KGstdLib
 ********************************************************************)

(* Checks ident on > 0 and formats string with two numbers *)
FUNCTION_BLOCK kgArLogWrite

	IF ident > 0 THEN

		_kgLogLine(sLoglineTemplate := text, lAttr1 := var1, lAttr2 := var2);

		_AsArLogWrite(enable := enable, ident := ident, logLevel := logLevel, errornr := errornr, mem := 0, len := 0, asciiString := _kgLogLine.pLogline);

		status := _AsArLogWrite.status;

	ELSE

		status := 1;

	END_IF

END_FUNCTION_BLOCK
```

#### kgRBcreate.st - Erzeuge Datenobjekt für Ringbuffer
```iecst
(********************************************************************
 * COPYRIGHT -- Herbert Kannegiesser GmbH
 ********************************************************************
 * Library: KGstdLib
 * File: kgRBcreate.st
 * Author: hunholz
 * Created: January 24, 2012
 ********************************************************************
 * Implementation of library KGstdLib
 ********************************************************************)

(* Erzeuge Datenobjekt für Ringbuffer *)
FUNCTION_BLOCK kgRBcreate

	_diRB.enable := TRUE;
	_diRB.pName := ADR(sName);
	_diRB();

	IF wCntEntry = 0 THEN

		wStatus := KG_ERR_RB_SIZE;
		RETURN;

	END_IF

	IF _diRB.status = ERR_OK THEN

		IF ((wCntEntry+1) * lLenEntry) > _diRB.len THEN

			_ddRB.enable := TRUE;
			_ddRB.ident := _diRB.ident;
			_ddRB();

			wPtrRead := 0;
			wPtrStart := 0;
			wPtrWrite := 0;

			IF _ddRB.status <> ERR_OK THEN

				wStatus := _ddRB.status;
				RETURN;

			END_IF

		END_IF

	END_IF

	_diRB();

	IF _diRB.status = doERR_MODULNOTFOUND  THEN

		wPtrRead := 0;
		wPtrStart := 0;
		wPtrWrite := 0;

		_dcRB.enable := TRUE;
		_dcRB.pName := ADR(sName);
		_dcRB.len := (wCntEntry+1) * lLenEntry;
		_dcRB.MemType := bMemType;
		_dcRB();

		IF _dcRB.status = ERR_OK OR _dcRB.status = doERR_DUPOBJECT  THEN

			_diRB();

			IF _diRB.status <> ERR_OK THEN

				wStatus := _diRB.status;
				RETURN;

			END_IF;

		ELSE

			wStatus := _diRB.status;
			RETURN;

		END_IF;

	ELSIF _diRB.status <> ERR_OK THEN

		wStatus := _diRB.status;
		RETURN;

	END_IF;

	doIdent := _diRB.ident;
	doLen := _diRB.len;
	pDatObjMem := _diRB.pDatObjMem;

	wStatus := ERR_OK;

END_FUNCTION_BLOCK
```

#### kgRBinsert.st - Insert any entry into a ringbuffer
```iecst
(********************************************************************
 * COPYRIGHT -- Herbert Kannegiesser GmbH
 ********************************************************************
 * Library: KGstdLib
 * File: kgRBinsert.st
 * Author: hunholz
 * Created: December 20, 2011
 ********************************************************************
 * Implementation of library KGstdLib
 ********************************************************************)

(* Insert any entry into a ringbuffer *)
FUNCTION_BLOCK kgRBinsert

	// VAR_IN_OUT UINT wPtrWrite
	// VAR_IN_OUT UINT wPtrRead
	// VAR_IN_OUT UINT wPtrStart
	// VAR_INPUT pEntry (Pointer to data)
	// VAR_INPUT lLenEntry (Size of data)
	// VAR_INPUT doLen
	// VAR_INPUT doIdent
	// VAR_OUT   wStatus

	_lRBlen := doLen / lLenEntry;

	// Der Ringbuffer muss wenigstens zwei Einträge halten können, wobei
	// ein Eintrag immer leer ist.
	IF _lRBlen <= 1 THEN
		wStatus := KG_ERR_RB_SIZE;
		RETURN;
	END_IF

	_wPtrMax := UDINT_TO_UINT(_lRBlen - 1);

	// Der Schreibzeiger muss immer auf eine gültige Position innerhalb des
	// Ringbuffers zeigen.
	IF  wPtrWrite > _wPtrMax THEN
		// Constant UINT KG_ERR_RB_WRITEPOINTER = 2 of KGstdLib
		wStatus := KG_ERR_RB_WRITEPOINTER;
		RETURN;
	END_IF;

	// Der Startzeiger muss immer auf eine gültige Position innerhalb des
	// Ringbuffers zeigen.
	IF  wPtrStart > _wPtrMax THEN
		// Constant UINT KG_ERR_RB_WRITEPOINTER = 2 of KGstdLib
		wStatus := KG_ERR_RB_STARTPOINTER;
		RETURN;
	END_IF;

	IF pEntry = 0 THEN
		// Constant UINT KG_ERR_RB_POINTER = 3 of KGstdLib
		wStatus := KG_ERR_RB_POINTER;
		RETURN;
	END_IF

	// VAR doWrite of DatObjWrite 'writes to a data object'
	// ADR() in ANSI C: &
	doWrite.enable := TRUE;			// enables execution
	doWrite.ident := doIdent;		// ID of the data object
	doWrite.len := lLenEntry;		// length of the data to be copied
	doWrite.Offset := wPtrWrite * lLenEntry;	// offset in the data area of the data object
	doWrite.pSource := pEntry;		// pointer to the data copied to the data object
	doWrite();

	IF doWrite.status = ERR_OK THEN

		wPtrWrite := UDINT_TO_UINT((wPtrWrite + 1) MOD _lRBlen);

		IF wPtrRead = wPtrWrite THEN
			wPtrRead := UDINT_TO_UINT((wPtrRead + 1) MOD _lRBlen);
		END_IF

		IF wPtrStart = wPtrWrite THEN
			wPtrStart := UDINT_TO_UINT((wPtrStart + 1) MOD _lRBlen);
		END_IF

	END_IF;

	wStatus := doWrite.status;	// UINT status: execution status: ERR_OK, ERR_FUB_ENABLE_FALSE, 0xXXXX = see help

END_FUNCTION_BLOCK
```

#### kgRBread.st - Reads one entry and moves the readpointer
```iecst
(********************************************************************
 * COPYRIGHT -- Herbert Kannegiesser GmbH
 ********************************************************************
 * Library: KGstdLib
 * File: kgRBread.st
 * Author: hunholz
 * Created: December 20, 2011
 ********************************************************************
 * Implementation of library KGstdLib
 ********************************************************************)

(* Reads one entry and moves the readpointer *)
FUNCTION_BLOCK kgRBread

	_lRBlen := doLen / lLenEntry;

	// Der Ringbuffer muss wenigstens zwei Einträge halten können, wobei
	// ein Eintrag immer leer ist.
	IF _lRBlen <= 1 THEN
		wStatus := KG_ERR_RB_SIZE;
		RETURN;
	END_IF

	_wPtrMax := UDINT_TO_UINT(_lRBlen - 1);

	// Der Schreibzeiger muss immer auf eine gültige Position innerhalb des
	// Ringbuffers zeigen.
	IF  wPtrWrite > _wPtrMax THEN
		// Constant UINT KG_ERR_RB_WRITEPOINTER = 2 of KGstdLib
		wStatus := KG_ERR_RB_WRITEPOINTER;
		RETURN;
	END_IF;

	// Der Startzeiger muss immer auf eine gültige Position innerhalb des
	// Ringbuffers zeigen.
	IF  wPtrRead > _wPtrMax THEN
		// Constant UINT KG_ERR_RB_WRITEPOINTER = 2 of KGstdLib
		wStatus := KG_ERR_RB_READPOINTER;
		RETURN;
	END_IF;

	IF (wPtrRead = wPtrWrite) THEN

		wStatus := KG_ERR_RB_NOREAD;
		RETURN;

	END_IF

	IF (wPtrRead > wPtrWrite) AND (UDINT_TO_UINT((wPtrWrite+1)MOD _lRBlen) <> wPtrStart) THEN
		// Lesezeiger zeigt in einen noch nicht beschriebenen Bereich
		wStatus := KG_ERR_RB_READPOINTER;
		RETURN;
	END_IF;

	IF (pEntry = 0) THEN

		wStatus := KG_ERR_RB_POINTER;
		RETURN;

	END_IF

	// doRead of DatObjRead 'reads from a data object'
	doRead.enable 		:= TRUE;	// enables execution
	doRead.ident 		:= doIdent;	// ID of the data object
	doRead.len 			:= lLenEntry;	// length of the data to be copied
	doRead.Offset 		:= wPtrRead * lLenEntry;	// offset in the data area of the data object
	doRead.pDestination := pEntry;	// memory to which the data to be read is copied
	doRead();

	IF doRead.status = ERR_OK THEN

		wPtrRead := UDINT_TO_UINT((wPtrRead + 1) MOD _lRBlen);

	END_IF

	wStatus := doRead.status; // executions status: ERR_OK, ERR_FUB_ENABLE_FALSE, 0xXXXX = see help

END_FUNCTION_BLOCK
```

#### kgRBloc.st - Free Readpointer access
```iecst
(********************************************************************
 * COPYRIGHT -- Herbert Kannegiesser GmbH
 ********************************************************************
 * Library: KGstdLib
 * File: kgRBloc.st
 * Author: hunholz
 * Created: December 20, 2011
 ********************************************************************
 * Implementation of library KGstdLib
 ********************************************************************)

(* Free Readpointer access *)
FUNCTION_BLOCK kgRBloc

	_lRBlen := doLen / lLenEntry;

	// Der Ringbuffer muss wenigstens zwei Einträge halten können, wobei
	// ein Eintrag immer leer ist.
	IF _lRBlen <= 1 THEN
		wStatus := KG_ERR_RB_SIZE;
		RETURN;
	END_IF

	_wPtrMax := UDINT_TO_UINT(_lRBlen - 1);

	IF ((wPtrWrite+1)MOD _lRBlen) = wPtrStart THEN
		_wActLen := _wPtrMax;
	ELSE
		_wActLen := wPtrWrite - wPtrStart;
	END_IF

	// Der Schreibzeiger muss immer auf eine gültige Position innerhalb des
	// Ringbuffers zeigen.
	IF  wPtrWrite > _wPtrMax THEN
		// Constant UINT KG_ERR_RB_WRITEPOINTER = 2 of KGstdLib
		wStatus := KG_ERR_RB_WRITEPOINTER;
		RETURN;
	END_IF;

	// Der Lesezeiger muss immer auf eine gültige Position innerhalb des
	// Ringbuffers zeigen.
	IF bMode = KG_RB_LOC_MODE_ABSOLUTE THEN

		IF  wPtrLoc > _wPtrMax THEN
			wStatus := KG_ERR_RB_LOCPOINTER;
			RETURN;
		END_IF;

	ELSIF wPtrLoc >= _wActLen THEN

		wStatus := KG_ERR_RB_LOCPOINTER;
		RETURN;

	END_IF

	_wPtrLoc := MUX(USINT_TO_SINT(bMode), wPtrLoc, UDINT_TO_UINT((wPtrStart+wPtrLoc)MOD _lRBlen), UDINT_TO_UINT((wPtrStart+(_wActLen - wPtrLoc - 1))MOD _lRBlen));

	IF (_wPtrLoc = wPtrWrite) THEN

		wStatus := KG_ERR_RB_NOREAD;
		RETURN;

	END_IF

	IF (_wPtrLoc > wPtrWrite) AND (UDINT_TO_UINT((wPtrWrite+1)MOD _lRBlen) <> wPtrStart) THEN
		// Lesezeiger zeigt in einen noch nicht beschriebenen Bereich
		wStatus := KG_ERR_RB_LOCPOINTER;
		RETURN;
	END_IF;

	IF (pEntry = 0) THEN

		wStatus := KG_ERR_RB_POINTER;
		RETURN;

	END_IF

	// doRead of DatObjRead 'reads from a data object'
	doRead.enable 			:= TRUE;	// enables execution
	doRead.ident 			:= doIdent;	// ID of the data object
	doRead.len 				:= lLenEntry * 1;	// length of the data to be copied
	doRead.Offset 			:= _wPtrLoc * lLenEntry;	// offset in the data area of the data object
	doRead.pDestination 	:= pEntry;	// memory to which the data to be read is copied
	doRead();

	wStatus := doRead.status; // executions status: ERR_OK, ERR_FUB_ENABLE_FALSE, 0xXXXX = see help

END_FUNCTION_BLOCK
```

#### kgGUIDisZero.st - Prüfen, ob alle 16 Byte der GUID 0 sind.
```iecst
(********************************************************************
 * COPYRIGHT -- Herbert Kannegiesser GmbH
 ********************************************************************
 * Library: KGstdLib
 * File: kgGUIDisZero.st
 * Author: hunholz
 * Created: January 03, 2012
 ********************************************************************
 * Implementation of library KGstdLib
 ********************************************************************)

(* Prüfen, ob alle 16 Byte der GUID 0 sind. *)
FUNCTION kgGUIDisZero

	_bGUID ACCESS ADR(GUID);

	kgGUIDisZero := TRUE;

	FOR _i := 0 TO 15 DO
		IF _bGUID[_i] > 0 THEN
			kgGUIDisZero := FALSE;
			EXIT;
		END_IF
	END_FOR

END_FUNCTION
```

#### kgRBbulkloc.st - Lese mehrere Einträge gleichzeitig in ein Array
```iecst
(********************************************************************
 * COPYRIGHT -- Herbert Kannegiesser GmbH
 ********************************************************************
 * Library: KGstdLib
 * File: kgRBbulkloc.st
 * Author: hunholz
 * Created: January 24, 2012
 ********************************************************************
 * Implementation of library KGstdLib
 ********************************************************************)

(* Lese mehrere Einträge gleichzeitig in ein Array *)
FUNCTION_BLOCK kgRBbulkloc

	_lRBlen := doLen / lLenEntry;

	// Der Ringbuffer muss wenigstens zwei Einträge halten können, wobei
	// ein Eintrag immer leer ist.
	IF _lRBlen <= 1 THEN
		wStatus := KG_ERR_RB_SIZE;
		RETURN;
	END_IF

	_wPtrMax := UDINT_TO_UINT(_lRBlen - 1);

	IF ((wPtrWrite+1)MOD _lRBlen) = wPtrStart THEN
		_wActLen := _wPtrMax;
	ELSE
		_wActLen := wPtrWrite - wPtrStart;
	END_IF

	// Der Schreibzeiger muss immer auf eine gültige Position innerhalb des
	// Ringbuffers zeigen.
	IF  wPtrWrite > _wPtrMax THEN
		// Constant UINT KG_ERR_RB_WRITEPOINTER = 2 of KGstdLib
		wStatus := KG_ERR_RB_WRITEPOINTER;
		RETURN;
	END_IF;

	// Der Lesezeiger muss immer auf eine gültige Position innerhalb des
	// Ringbuffers zeigen.
	IF bMode = KG_RB_LOC_MODE_ABSOLUTE THEN

		IF  wPtrLoc > _wPtrMax THEN
			wStatus := KG_ERR_RB_LOCPOINTER;
			RETURN;
		END_IF;

	ELSIF wPtrLoc >= _wActLen THEN

		wStatus := KG_ERR_RB_LOCPOINTER;
		RETURN;

	END_IF

	_wPtrLoc := MUX(USINT_TO_SINT(bMode), wPtrLoc, UDINT_TO_UINT((wPtrStart+wPtrLoc)MOD _lRBlen), UDINT_TO_UINT((wPtrStart+(_wActLen - wPtrLoc - 1))MOD _lRBlen));

	IF (_wPtrLoc = wPtrWrite) THEN

		wStatus := KG_ERR_RB_NOREAD;
		RETURN;

	END_IF

	IF (_wPtrLoc > wPtrWrite) AND (UDINT_TO_UINT((wPtrWrite+1)MOD _lRBlen) <> wPtrStart) THEN
		// Lesezeiger zeigt in einen noch nicht beschriebenen Bereich
		wStatus := KG_ERR_RB_LOCPOINTER;
		RETURN;
	END_IF;

	IF (pEntry = 0) THEN

		wStatus := KG_ERR_RB_POINTER;
		RETURN;

	END_IF

	wCntLoc := 0;

	brsmemset(pEntry, 0, lLenEntry*wCntEntry);

	IF (wCntEntry = 0) THEN

		wStatus := ERR_OK;
		RETURN;

	END_IF

	FOR _i := 0 TO wCntEntry-1 DO

		// doRead of DatObjRead 'reads from a data object'
		_doRead.enable 			:= TRUE;	// enables execution
		_doRead.ident 			:= doIdent;	// ID of the data object
		_doRead.len 				:= lLenEntry * 1;	// length of the data to be copied
		_doRead.Offset 			:= _wPtrLoc * lLenEntry;	// offset in the data area of the data object
		_doRead.pDestination 	:= pEntry + (_i * lLenEntry);	// memory to which the data to be read is copied
		_doRead();

		wStatus := _doRead.status; // executions status: ERR_OK, ERR_FUB_ENABLE_FALSE, 0xXXXX = see help

		IF wStatus <> ERR_OK THEN
			RETURN;
		END_IF

		wCntLoc := wCntLoc + 1;

		IF bMode = KG_RB_LOC_MODE_FROMEND THEN

			IF _wPtrLoc = wPtrStart THEN
				RETURN;
			END_IF

			IF _wPtrLoc = 0 THEN
				_wPtrLoc := UDINT_TO_UINT(_lRBlen);
			END_IF

			_wPtrLoc := _wPtrLoc - 1;

		ELSE

			_wPtrLoc := UDINT_TO_UINT((_wPtrLoc + 1) MOD _lRBlen);

			IF _wPtrLoc = wPtrWrite THEN
				RETURN;
			END_IF

		END_IF

	END_FOR

END_FUNCTION_BLOCK
```

#### kgGetEthPort.st - Returns the CPUs ethernet port as string
```iecst
(********************************************************************
 * COPYRIGHT -- Microsoft
 ********************************************************************
 * Library: Netlink
 * File: GetEthPort.st
 * Author: hunholz
 * Created: June 30, 2011
 ********************************************************************
 * Implementation of library Netlink
 ********************************************************************)

(* Returns the CPUs ethernet port as string *)
FUNCTION_BLOCK kgGetEthPort

	IF enable THEN

		IF adrIF <= 16#3FFF THEN

			_bStep := 10;
			status := KG_ERR_GETETHPORT_ADRIF;
			RETURN;

		END_IF

		_xReady := FALSE;

		REPEAT

			CASE (_bStep) OF

				10:
				// Create Info
					DiagCreateInfo_CPU(enable := TRUE, infoKind := asdiagPLUGGED);

					status := DiagCreateInfo_CPU.status;

					IF (status = ERR_OK) THEN
			  			_bStep := 12;
					END_IF;

				12:
					// Get Info
					DiagGetNumInfo_CPU(enable := TRUE,
											ident := DiagCreateInfo_CPU.ident,
											index := 0,
											infoCode := asdiagPLUGGED_MODNO);

					status := DiagGetNumInfo_CPU.status;

					IF (status = ERR_OK) THEN

						CASE DiagGetNumInfo_CPU.value OF

							KG_CPU_X20CP1484, KG_CPU_X20CP1484_1, KG_CPU_X20CP3484_1, KG_CPU_X20CP1486, KG_CPU_X20CP3486, KG_CPU_X20CP3585, KG_CPU_X20CP1584,KG_CPU_X20CP1586, KG_CPU_X20CP3484:
								brsstrcpy(adrIF, ADR('IF2'));

							KG_CPU_PP420_1043_75, KG_CPU_CTT_11, KG_CPU_PP65_0571_P74, KG_CPU_PCT_04, KG_CPU_PCT_03:
								brsstrcpy(adrIF, ADR('IF5'));

							ELSE	// keinen gültigen B&R ID-Code gefunden
								brsstrcpy(adrIF, ADR('IF3'));
								//status := KG_ERR_GETETHPORT_IFSTRING;

						END_CASE

						_bStep := 14;

					ELSIF (status <> ERR_FUB_BUSY) THEN
						_bStep := 10;
					END_IF;

				14:
					// Write string to variable

					DiagDisposeInfo_CPU(enable := TRUE, ident := DiagCreateInfo_CPU.ident);

					status := DiagDisposeInfo_CPU.status;

					_xReady := (status = ERR_OK);

					IF (status <> ERR_FUB_BUSY) THEN

						_bStep := 10;
						DiagCreateInfo_CPU(enable := FALSE);
						DiagDisposeInfo_CPU(enable := FALSE);
						DiagGetNumInfo_CPU(enable := FALSE);

					END_IF;

				ELSE

					_bStep := 10;
					status := ERR_FUB_BUSY;

			END_CASE;

			UNTIL

			status <> ERR_OK OR _xReady

		END_REPEAT

	ELSE

		status := ERR_FUB_ENABLE_FALSE;
		_bStep := 10;

	END_IF

END_FUNCTION_BLOCK
```

#### kgGetLineNumberW3.st - Maschinennummer und -typ aus Stationsadresse berechnen
```iecst
(********************************************************************
 * COPYRIGHT -- Herbert Kannegiesser GmbH
 ********************************************************************
 * Library: KGstdLib
 * File: kgGetLineNumberW3.st
 * Author: hunholz
 * Created: January 27, 2012
 * Changed: February 8, 2012
 ********************************************************************
 * Implementation of library KGstdLib
 ********************************************************************)

(* Liniennummer und -typ aus Stationsadresse berechnen *)
FUNCTION kgGetLineNumberW3

	_MachineType ACCESS pMachineType;

	_MachineType := kgW3NOTDEFINED;
	kgGetLineNumberW3 := 0;

	CASE Station OF

		1..10:
			kgGetLineNumberW3 := Station;
			_MachineType := kgW3LOADSYSTEM;

		11..30:
			kgGetLineNumberW3 := Station - 10;
			_MachineType := kgW3WASHER;

		31..40:
			kgGetLineNumberW3 := Station - 30;
			_MachineType := kgW3WETSHUTTLE;

		41..50:
			kgGetLineNumberW3 := Station - 40;
			_MachineType := kgW3EXTRACTOR;

		51..60:
			kgGetLineNumberW3 := Station - 50;
			_MachineType := kgW3EXTRACTOR2;

		61..70:
			kgGetLineNumberW3 := Station - 60;
			_MachineType := kgW3CONVEYOR;

		71..100:
			kgGetLineNumberW3 := Station - 70;
			_MachineType := kgW3DRYER;

		111..120:
			kgGetLineNumberW3 := Station - 110;
			_MachineType := kgW3SHAKER;

		121..150:
			kgGetLineNumberW3 := Station - 120;
			_MachineType := kgW3SINGLEWASHER;

		151..160:
			kgGetLineNumberW3 := Station - 150;
			_MachineType := kgW3PROCESS;

		161..180:
			kgGetLineNumberW3 := Station - 160;
			_MachineType := kgW3IFBOX;

		181..200:
			kgGetLineNumberW3 := Station - 180;
			_MachineType := kgW3DEVICE;

		202:
			kgGetLineNumberW3 := 202;
			_MachineType := kgW3SERVER;

		211..230:
			kgGetLineNumberW3 := Station - 210;
			_MachineType := kgW3PCSTATION;

		231..250:
			kgGetLineNumberW3 := Station - 230;
			_MachineType := kgW3BIT;

	END_CASE

END_FUNCTION
```
